LIN {X 0,Y 590.788,Z 779.363,A -85,B 0,C 180,E1 25957.461,E2 25957.461} C_VEL
LIN {X 0,Y 599.136,Z 539.916,A -85,B 0,C 180,E1 25954.035,E2 25954.035} C_VEL
LIN {X 0,Y 604.278,Z 401.411,A -85,B 0,C 180,E1 25952.028,E2 25952.028} C_VEL
LIN {X 0,Y 593.567,Z 385.03,A -85,B 0,C 180,E1 25950.244,E2 25950.244} C_VEL
LIN {X 0,Y 582.771,Z 369.958,A -85,B 0,C 180,E1 25948.293,E2 25948.293} C_VEL
LIN {X 0,Y 574.753,Z 359.34,A -85,B 0,C 180,E1 25946.725,E2 25946.725} C_VEL
LIN {X 0,Y 565.367,Z 346.989,A -85,B 0,C 180,E1 25944.67,E2 25944.67} C_VEL
LIN {X 0,Y 561.776,Z 340.566,A -85,B 0,C 180,E1 25943.052,E2 25943.052} C_VEL
LIN {X 0,Y 559.747,Z 336.589,A -85,B 0,C 180,E1 25942.032,E2 25942.032} C_VEL
LIN {X 0,Y 557.15,Z 331.806,A -85,B 0,C 180,E1 25940.705,E2 25940.705} C_VEL
LIN {X 0,Y 555.047,Z 327.971,A -85,B 0,C 180,E1 25939.577,E2 25939.577} C_VEL
LIN {X 0,Y 552.236,Z 323.289,A -85,B 0,C 180,E1 25938.036,E2 25938.036} C_VEL
LIN {X 0,Y 551.411,Z 321.689,A -85,B 0,C 180,E1 25937.519,E2 25937.519} C_VEL
LIN {X 0,Y 549.142,Z 318.092,A -85,B 0,C 180,E1 25936.176,E2 25936.176} C_VEL
LIN {X 0,Y 548.449,Z 316.544,A -85,B 0,C 180,E1 25935.654,E2 25935.654} C_VEL
LIN {X 0,Y 545.984,Z 313.041,A -85,B 0,C 180,E1 25934.097,E2 25934.097} C_VEL
LIN {X 0,Y 545.58,Z 311.452,A -85,B 0,C 180,E1 25933.459,E2 25933.459} C_VEL
LIN {X 0,Y 545.545,Z 311.25,A -85,B 0,C 180,E1 25930.241,E2 25930.241} C_VEL
LIN {X 0,Y 545.551,Z 311.212,A -85,B 0,C 180,E1 25926.842,E2 25926.842} C_VEL
LIN {X 0,Y 545.55,Z 311.247,A -85,B 0,C 180,E1 25923.362,E2 25923.362} C_VEL
LIN {X 0,Y 545.546,Z 311.235,A -85,B 0,C 180,E1 25920,E2 25920} C_VEL
LIN {X 0,Y 545.545,Z 311.216,A -85,B 0,C 180,E1 25916.743,E2 25916.743} C_VEL
LIN {X 0,Y 545.564,Z 311.275,A -85,B 0,C 180,E1 25913.264,E2 25913.264} C_VEL
LIN {X 0,Y 545.547,Z 311.219,A -85,B 0,C 180,E1 25909.799,E2 25909.799} C_VEL
LIN {X 0,Y 545.543,Z 311.229,A -85,B 0,C 180,E1 25906.54,E2 25906.54} C_VEL
LIN {X 0,Y 545.559,Z 311.26,A -85,B 0,C 180,E1 25903.167,E2 25903.167} C_VEL
LIN {X 0,Y 545.63,Z 311.708,A -85,B 0,C 180,E1 25901.945,E2 25901.945} C_VEL
LIN {X 0,Y 547.322,Z 315.338,A -85,B 0,C 180,E1 25900.58,E2 25900.58} C_VEL
LIN {X 0,Y 549.044,Z 317.373,A -85,B 0,C 180,E1 25899.645,E2 25899.645} C_VEL
LIN {X 0,Y 551.001,Z 321.182,A -85,B 0,C 180,E1 25898.384,E2 25898.384} C_VEL
LIN {X 0,Y 552.44,Z 323.078,A -85,B 0,C 180,E1 25897.661,E2 25897.661} C_VEL
LIN {X 0,Y 554.498,Z 326.812,A -85,B 0,C 180,E1 25896.515,E2 25896.515} C_VEL
LIN {X 0,Y 555.592,Z 328.37,A -85,B 0,C 180,E1 25896,E2 25896} C_VEL
LIN {X 0,Y 557.889,Z 332.375,A -85,B 0,C 180,E1 25894.864,E2 25894.864} C_VEL
LIN {X 0,Y 561.672,Z 339.042,A -85,B 0,C 180,E1 25893.107,E2 25893.107} C_VEL
LIN {X 0,Y 564.696,Z 344.498,A -85,B 0,C 180,E1 25891.786,E2 25891.786} C_VEL
LIN {X 0,Y 567.543,Z 349.518,A -85,B 0,C 180,E1 25890.674,E2 25890.674} C_VEL
LIN {X 0,Y 578.522,Z 363.571,A -85,B 0,C 180,E1 25888.391,E2 25888.391} C_VEL
LIN {X 0,Y 590.148,Z 379.589,A -85,B 0,C 180,E1 25886.239,E2 25886.239} C_VEL
LIN {X 0,Y 600.117,Z 394.544,A -85,B 0,C 180,E1 25884.532,E2 25884.532} C_VEL
LIN {X 0,Y 607.718,Z 406.774,A -85,B 0,C 180,E1 25883.311,E2 25883.311} C_VEL
LIN {X 0,Y 600.499,Z 616.97,A -85,B 0,C 180,E1 25880.226,E2 25880.226} C_VEL
LIN {X 0,Y 594.04,Z 824.716,A -85,B 0,C 180,E1 25877.25,E2 25877.25} C_VEL
LIN {X 0,Y 592.323,Z 852.282,A -85,B 0,C 180,E1 25876.741,E2 25876.741} C_VEL
LIN {X 0,Y 590.04,Z 878.41,A -85,B 0,C 180,E1 25876.074,E2 25876.074} C_VEL
LIN {X 0,Y 587.877,Z 899.594,A -85,B 0,C 180,E1 25875.411,E2 25875.411} C_VEL
LIN {X 0,Y 585.51,Z 920.264,A -85,B 0,C 180,E1 25874.645,E2 25874.645} C_VEL
LIN {X 0,Y 582.87,Z 941.326,A -85,B 0,C 180,E1 25873.734,E2 25873.734} C_VEL
LIN {X 0,Y 579.321,Z 967.03,A -85,B 0,C 180,E1 25872.441,E2 25872.441} C_VEL
LIN {X 0,Y 575.836,Z 989.761,A -85,B 0,C 180,E1 25871.096,E2 25871.096} C_VEL
LIN {X 0,Y 572.812,Z 1008.617,A -85,B 0,C 180,E1 25869.837,E2 25869.837} C_VEL
LIN {X 0,Y 569.828,Z 1026.571,A -85,B 0,C 180,E1 25868.5,E2 25868.5} C_VEL
LIN {X 0,Y 566.727,Z 1044.849,A -85,B 0,C 180,E1 25866.986,E2 25866.986} C_VEL
LIN {X 0,Y 564.355,Z 1058.093,A -85,B 0,C 180,E1 25865.761,E2 25865.761} C_VEL
LIN {X 0,Y 561.301,Z 1074.316,A -85,B 0,C 180,E1 25864.071,E2 25864.071} C_VEL
LIN {X 0,Y 557.893,Z 1092.847,A -85,B 0,C 180,E1 25861.918,E2 25861.918} C_VEL
LIN {X 0,Y 554.675,Z 1110.292,A -85,B 0,C 180,E1 25859.598,E2 25859.598} C_VEL
LIN {X 0,Y 552.277,Z 1124.437,A -85,B 0,C 180,E1 25857.483,E2 25857.483} C_VEL
LIN {X 0,Y 550.164,Z 1137.628,A -85,B 0,C 180,E1 25855.283,E2 25855.283} C_VEL
LIN {X 0,Y 548.084,Z 1152.164,A -85,B 0,C 180,E1 25852.526,E2 25852.526} C_VEL
LIN {X 0,Y 546.633,Z 1163.604,A -85,B 0,C 180,E1 25850.002,E2 25850.002} C_VEL
LIN {X 0,Y 545.65,Z 1172.702,A -85,B 0,C 180,E1 25847.709,E2 25847.709} C_VEL
LIN {X 0,Y 544.935,Z 1180.92,A -85,B 0,C 180,E1 25845.32,E2 25845.32} C_VEL
LIN {X 0,Y 544.377,Z 1189.025,A -85,B 0,C 180,E1 25842.517,E2 25842.517} C_VEL
LIN {X 0,Y 544.091,Z 1195.291,A -85,B 0,C 180,E1 25839.734,E2 25839.734} C_VEL
LIN {X 0,Y 543.978,Z 1199.369,A -85,B 0,C 180,E1 25837.392,E2 25837.392} C_VEL
LIN {X 0,Y 543.924,Z 1202.439,A -85,B 0,C 180,E1 25834.956,E2 25834.956} C_VEL
LIN {X 0,Y 543.91,Z 1204.495,A -85,B 0,C 180,E1 25832.212,E2 25832.212} C_VEL
LIN {X 0,Y 543.894,Z 1204.894,A -85,B 0,C 180,E1 25829.473,E2 25829.473} C_VEL
LIN {X 0,Y 543.915,Z 1204.043,A -85,B 0,C 180,E1 25827.05,E2 25827.05} C_VEL
LIN {X 0,Y 543.93,Z 1202.097,A -85,B 0,C 180,E1 25824.727,E2 25824.727} C_VEL
LIN {X 0,Y 543.984,Z 1198.889,A -85,B 0,C 180,E1 25822.289,E2 25822.289} C_VEL
LIN {X 0,Y 544.153,Z 1193.819,A -85,B 0,C 180,E1 25819.519,E2 25819.519} C_VEL
LIN {X 0,Y 544.513,Z 1186.94,A -85,B 0,C 180,E1 25816.717,E2 25816.717} C_VEL
LIN {X 0,Y 545.002,Z 1179.859,A -85,B 0,C 180,E1 25814.355,E2 25814.355} C_VEL
LIN {X 0,Y 545.737,Z 1171.893,A -85,B 0,C 180,E1 25812.074,E2 25812.074} C_VEL
LIN {X 0,Y 546.863,Z 1161.773,A -85,B 0,C 180,E1 25809.561,E2 25809.561} C_VEL
LIN {X 0,Y 548.605,Z 1148.289,A -85,B 0,C 180,E1 25806.703,E2 25806.703} C_VEL
LIN {X 0,Y 550.465,Z 1135.727,A -85,B 0,C 180,E1 25804.386,E2 25804.386} C_VEL
LIN {X 0,Y 552.556,Z 1122.677,A -85,B 0,C 180,E1 25802.238,E2 25802.238} C_VEL
LIN {X 0,Y 555.576,Z 1105.587,A -85,B 0,C 180,E1 25799.741,E2 25799.741} C_VEL
LIN {X 0,Y 558.686,Z 1088.219,A -85,B 0,C 180,E1 25797.527,E2 25797.527} C_VEL
LIN {X 0,Y 561.576,Z 1072.791,A -85,B 0,C 180,E1 25795.763,E2 25795.763} C_VEL
LIN {X 0,Y 564.688,Z 1056.271,A -85,B 0,C 180,E1 25794.058,E2 25794.058} C_VEL
LIN {X 0,Y 567.368,Z 1041.067,A -85,B 0,C 180,E1 25792.683,E2 25792.683} C_VEL
LIN {X 0,Y 571.091,Z 1019.418,A -85,B 0,C 180,E1 25790.929,E2 25790.929} C_VEL
LIN {X 0,Y 574.899,Z 996.123,A -85,B 0,C 180,E1 25789.293,E2 25789.293} C_VEL
LIN {X 0,Y 578.011,Z 976.204,A -85,B 0,C 180,E1 25788.061,E2 25788.061} C_VEL
LIN {X 0,Y 580.949,Z 956.254,A -85,B 0,C 180,E1 25786.968,E2 25786.968} C_VEL
LIN {X 0,Y 583.868,Z 935.058,A -85,B 0,C 180,E1 25785.952,E2 25785.952} C_VEL
LIN {X 0,Y 587.105,Z 909.113,A -85,B 0,C 180,E1 25784.89,E2 25784.89} C_VEL
LIN {X 0,Y 589.775,Z 883.656,A -85,B 0,C 180,E1 25784.048,E2 25784.048} C_VEL
LIN {X 0,Y 591.743,Z 862.08,A -85,B 0,C 180,E1 25783.464,E2 25783.464} C_VEL
LIN {X 0,Y 593.379,Z 840.414,A -85,B 0,C 180,E1 25782.996,E2 25782.996} C_VEL
LIN {X 0,Y 594.742,Z 814.677,A -85,B 0,C 180,E1 25782.568,E2 25782.568} C_VEL
LIN {X 0,Y 601.152,Z 593.035,A -85,B 0,C 180,E1 25779.439,E2 25779.439} C_VEL
LIN {X 0,Y 606.786,Z 406.521,A -85,B 0,C 180,E1 25776.755,E2 25776.755} C_VEL
LIN {X 0,Y 589.939,Z 382.189,A -85,B 0,C 180,E1 25774.39,E2 25774.39} C_VEL
LIN {X 0,Y 573.518,Z 359.446,A -85,B 0,C 180,E1 25771.888,E2 25771.888} C_VEL
LIN {X 0,Y 565.896,Z 348.958,A -85,B 0,C 180,E1 25770.589,E2 25770.589} C_VEL
LIN {X 0,Y 558.763,Z 335.53,A -85,B 0,C 180,E1 25768.192,E2 25768.192} C_VEL
LIN {X 0,Y 553.373,Z 325.76,A -85,B 0,C 180,E1 25766.276,E2 25766.276} C_VEL
LIN {X 0,Y 550.642,Z 320.898,A -85,B 0,C 180,E1 25765.26,E2 25765.26} C_VEL
LIN {X 0,Y 548.552,Z 317.065,A -85,B 0,C 180,E1 25764.442,E2 25764.442} C_VEL
LIN {X 0,Y 545.84,Z 312.595,A -85,B 0,C 180,E1 25763.405,E2 25763.405} C_VEL
LIN {X 0,Y 545.574,Z 311.357,A -85,B 0,C 180,E1 25763.074,E2 25763.074} C_VEL
LIN {X 0,Y 545.549,Z 311.245,A -85,B 0,C 180,E1 25759.709,E2 25759.709} C_VEL
LIN {X 0,Y 545.543,Z 311.204,A -85,B 0,C 180,E1 25756.395,E2 25756.395} C_VEL
LIN {X 0,Y 545.559,Z 311.271,A -85,B 0,C 180,E1 25753.028,E2 25753.028} C_VEL
LIN {X 0,Y 545.55,Z 311.196,A -85,B 0,C 180,E1 25749.592,E2 25749.592} C_VEL
LIN {X 0,Y 545.544,Z 311.275,A -85,B 0,C 180,E1 25746.208,E2 25746.208} C_VEL
LIN {X 0,Y 545.559,Z 311.277,A -85,B 0,C 180,E1 25742.77,E2 25742.77} C_VEL
LIN {X 0,Y 545.566,Z 311.272,A -85,B 0,C 180,E1 25739.37,E2 25739.37} C_VEL
LIN {X 0,Y 545.539,Z 311.278,A -85,B 0,C 180,E1 25736.006,E2 25736.006} C_VEL
LIN {X 0,Y 545.565,Z 311.267,A -85,B 0,C 180,E1 25732.629,E2 25732.629} C_VEL
LIN {X 0,Y 545.558,Z 311.268,A -85,B 0,C 180,E1 25729.216,E2 25729.216} C_VEL
LIN {X 0,Y 545.534,Z 311.267,A -85,B 0,C 180,E1 25725.825,E2 25725.825} C_VEL
LIN {X 0,Y 545.563,Z 311.258,A -85,B 0,C 180,E1 25722.508,E2 25722.508} C_VEL
LIN {X 0,Y 545.545,Z 311.261,A -85,B 0,C 180,E1 25719.172,E2 25719.172} C_VEL
LIN {X 0,Y 545.527,Z 311.212,A -85,B 0,C 180,E1 25715.759,E2 25715.759} C_VEL
LIN {X 0,Y 545.566,Z 311.254,A -85,B 0,C 180,E1 25712.374,E2 25712.374} C_VEL
LIN {X 0,Y 545.524,Z 311.209,A -85,B 0,C 180,E1 25709.067,E2 25709.067} C_VEL
LIN {X 0,Y 545.531,Z 311.278,A -85,B 0,C 180,E1 25705.565,E2 25705.565} C_VEL
LIN {X 0,Y 545.573,Z 311.483,A -85,B 0,C 180,E1 25702.673,E2 25702.673} C_VEL
LIN {X 0,Y 547.112,Z 315.058,A -85,B 0,C 180,E1 25701.85,E2 25701.85} C_VEL
LIN {X 0,Y 548.285,Z 316.8,A -85,B 0,C 180,E1 25701.413,E2 25701.413} C_VEL
LIN {X 0,Y 550.113,Z 320.411,A -85,B 0,C 180,E1 25700.628,E2 25700.628} C_VEL
LIN {X 0,Y 551.214,Z 322.439,A -85,B 0,C 180,E1 25700.183,E2 25700.183} C_VEL
LIN {X 0,Y 554.259,Z 328.328,A -85,B 0,C 180,E1 25698.954,E2 25698.954} C_VEL
LIN {X 0,Y 556.098,Z 331.679,A -85,B 0,C 180,E1 25698.259,E2 25698.259} C_VEL
LIN {X 0,Y 562.517,Z 344.33,A -85,B 0,C 180,E1 25695.83,E2 25695.83} C_VEL
LIN {X 0,Y 564.644,Z 348.18,A -85,B 0,C 180,E1 25695.187,E2 25695.187} C_VEL
LIN {X 0,Y 579.441,Z 368.707,A -85,B 0,C 180,E1 25692.811,E2 25692.811} C_VEL
LIN {X 0,Y 594.651,Z 390.663,A -85,B 0,C 180,E1 25690.574,E2 25690.574} C_VEL
LIN {X 0,Y 601.282,Z 400.794,A -85,B 0,C 180,E1 25689.652,E2 25689.652} C_VEL
LIN {X 0,Y 594.576,Z 614.61,A -85,B 0,C 180,E1 25686.64,E2 25686.64} C_VEL
LIN {X 0,Y 593.661,Z 622.309,A -85,B 0,C 180,E1 25686.601,E2 25686.601} C_VEL
LIN {X 0,Y 588.726,Z 642.915,A -85,B 0,C 180,E1 25686.752,E2 25686.752} C_VEL
LIN {X 0,Y 587.972,Z 649.525,A -85,B 0,C 180,E1 25686.715,E2 25686.715} C_VEL
LIN {X 0,Y 583.597,Z 784.855,A -85,B 0,C 180,E1 25684.797,E2 25684.797} C_VEL
LIN {X 0,Y 581.939,Z 811.482,A -85,B 0,C 180,E1 25684.279,E2 25684.279} C_VEL
LIN {X 0,Y 579.838,Z 835.361,A -85,B 0,C 180,E1 25683.639,E2 25683.639} C_VEL
LIN {X 0,Y 577.586,Z 856.724,A -85,B 0,C 180,E1 25682.927,E2 25682.927} C_VEL
LIN {X 0,Y 574.452,Z 882.144,A -85,B 0,C 180,E1 25681.887,E2 25681.887} C_VEL
LIN {X 0,Y 571.387,Z 903.281,A -85,B 0,C 180,E1 25680.845,E2 25680.845} C_VEL
LIN {X 0,Y 568.337,Z 922.57,A -85,B 0,C 180,E1 25679.743,E2 25679.743} C_VEL
LIN {X 0,Y 564.588,Z 944.778,A -85,B 0,C 180,E1 25678.277,E2 25678.277} C_VEL
LIN {X 0,Y 560.871,Z 964.796,A -85,B 0,C 180,E1 25676.727,E2 25676.727} C_VEL
LIN {X 0,Y 557.656,Z 981.532,A -85,B 0,C 180,E1 25675.26,E2 25675.26} C_VEL
LIN {X 0,Y 553.995,Z 1000.37,A -85,B 0,C 180,E1 25673.394,E2 25673.394} C_VEL
LIN {X 0,Y 550.34,Z 1018.522,A -85,B 0,C 180,E1 25671.307,E2 25671.307} C_VEL
LIN {X 0,Y 547.515,Z 1033.091,A -85,B 0,C 180,E1 25669.412,E2 25669.412} C_VEL
LIN {X 0,Y 544.571,Z 1048.925,A -85,B 0,C 180,E1 25667.084,E2 25667.084} C_VEL
LIN {X 0,Y 542.122,Z 1062.63,A -85,B 0,C 180,E1 25664.745,E2 25664.745} C_VEL
LIN {X 0,Y 540.353,Z 1073.663,A -85,B 0,C 180,E1 25662.612,E2 25662.612} C_VEL
LIN {X 0,Y 538.583,Z 1086.085,A -85,B 0,C 180,E1 25659.834,E2 25659.834} C_VEL
LIN {X 0,Y 537.402,Z 1096.194,A -85,B 0,C 180,E1 25657.161,E2 25657.161} C_VEL
LIN {X 0,Y 536.685,Z 1105.073,A -85,B 0,C 180,E1 25654.488,E2 25654.488} C_VEL
LIN {X 0,Y 536.258,Z 1111.875,A -85,B 0,C 180,E1 25651.923,E2 25651.923} C_VEL
LIN {X 0,Y 536.038,Z 1116.676,A -85,B 0,C 180,E1 25649.679,E2 25649.679} C_VEL
LIN {X 0,Y 535.95,Z 1120.549,A -85,B 0,C 180,E1 25647.327,E2 25647.327} C_VEL
LIN {X 0,Y 535.903,Z 1123.56,A -85,B 0,C 180,E1 25644.54,E2 25644.54} C_VEL
LIN {X 0,Y 535.915,Z 1124.748,A -85,B 0,C 180,E1 25642.172,E2 25642.172} C_VEL
LIN {X 0,Y 535.897,Z 1124.806,A -85,B 0,C 180,E1 25640.008,E2 25640.008} C_VEL
LIN {X 0,Y 535.914,Z 1123.784,A -85,B 0,C 180,E1 25637.72,E2 25637.72} C_VEL
LIN {X 0,Y 535.927,Z 1121.277,A -85,B 0,C 180,E1 25635.08,E2 25635.08} C_VEL
LIN {X 0,Y 536.034,Z 1117.021,A -85,B 0,C 180,E1 25632.412,E2 25632.412} C_VEL
LIN {X 0,Y 536.241,Z 1112.285,A -85,B 0,C 180,E1 25630.163,E2 25630.163} C_VEL
LIN {X 0,Y 536.603,Z 1106.05,A -85,B 0,C 180,E1 25627.775,E2 25627.775} C_VEL
LIN {X 0,Y 537.359,Z 1096.738,A -85,B 0,C 180,E1 25624.898,E2 25624.898} C_VEL
LIN {X 0,Y 538.514,Z 1086.699,A -85,B 0,C 180,E1 25622.223,E2 25622.223} C_VEL
LIN {X 0,Y 540.316,Z 1074.141,A -85,B 0,C 180,E1 25619.375,E2 25619.375} C_VEL
LIN {X 0,Y 542.16,Z 1062.795,A -85,B 0,C 180,E1 25617.167,E2 25617.167} C_VEL
LIN {X 0,Y 544.698,Z 1048.834,A -85,B 0,C 180,E1 25614.774,E2 25614.774} C_VEL
LIN {X 0,Y 547.719,Z 1032.714,A -85,B 0,C 180,E1 25612.4,E2 25612.4} C_VEL
LIN {X 0,Y 550.595,Z 1018.237,A -85,B 0,C 180,E1 25610.517,E2 25610.517} C_VEL
LIN {X 0,Y 554.342,Z 999.904,A -85,B 0,C 180,E1 25608.413,E2 25608.413} C_VEL
LIN {X 0,Y 557.857,Z 982.219,A -85,B 0,C 180,E1 25606.65,E2 25606.65} C_VEL
LIN {X 0,Y 561.158,Z 965.503,A -85,B 0,C 180,E1 25605.168,E2 25605.168} C_VEL
LIN {X 0,Y 565.097,Z 945.093,A -85,B 0,C 180,E1 25603.568,E2 25603.568} C_VEL
LIN {X 0,Y 569.057,Z 922.587,A -85,B 0,C 180,E1 25602.068,E2 25602.068} C_VEL
LIN {X 0,Y 572.335,Z 902.847,A -85,B 0,C 180,E1 25600.93,E2 25600.93} C_VEL
LIN {X 0,Y 576.001,Z 878.581,A -85,B 0,C 180,E1 25599.737,E2 25599.737} C_VEL
LIN {X 0,Y 578.96,Z 855.49,A -85,B 0,C 180,E1 25598.807,E2 25598.807} C_VEL
LIN {X 0,Y 581.4,Z 833.425,A -85,B 0,C 180,E1 25598.073,E2 25598.073} C_VEL
LIN {X 0,Y 583.848,Z 805.824,A -85,B 0,C 180,E1 25597.362,E2 25597.362} C_VEL
LIN {X 0,Y 585.261,Z 783.212,A -85,B 0,C 180,E1 25596.937,E2 25596.937} C_VEL
LIN {X 0,Y 593.876,Z 548.322,A -85,B 0,C 180,E1 25593.549,E2 25593.549} C_VEL
LIN {X 0,Y 599.32,Z 405.367,A -85,B 0,C 180,E1 25591.452,E2 25591.452} C_VEL
LIN {X 0,Y 589.748,Z 390.74,A -85,B 0,C 180,E1 25589.815,E2 25589.815} C_VEL
LIN {X 0,Y 579.93,Z 376.804,A -85,B 0,C 180,E1 25587.996,E2 25587.996} C_VEL
LIN {X 0,Y 571.777,Z 365.901,A -85,B 0,C 180,E1 25586.371,E2 25586.371} C_VEL
LIN {X 0,Y 561.894,Z 353.19,A -85,B 0,C 180,E1 25584.216,E2 25584.216} C_VEL
LIN {X 0,Y 557.113,Z 347.152,A -85,B 0,C 180,E1 25583.033,E2 25583.033} C_VEL
LIN {X 0,Y 554.637,Z 342.483,A -85,B 0,C 180,E1 25581.8,E2 25581.8} C_VEL
LIN {X 0,Y 552.29,Z 338.046,A -85,B 0,C 180,E1 25580.562,E2 25580.562} C_VEL
LIN {X 0,Y 549.649,Z 333.261,A -85,B 0,C 180,E1 25579.114,E2 25579.114} C_VEL
LIN {X 0,Y 547.469,Z 329.509,A -85,B 0,C 180,E1 25577.869,E2 25577.869} C_VEL
LIN {X 0,Y 546.617,Z 327.981,A -85,B 0,C 180,E1 25577.348,E2 25577.348} C_VEL
LIN {X 0,Y 544.451,Z 324.327,A -85,B 0,C 180,E1 25575.991,E2 25575.991} C_VEL
LIN {X 0,Y 543.712,Z 322.903,A -85,B 0,C 180,E1 25575.465,E2 25575.465} C_VEL
LIN {X 0,Y 541.474,Z 319.601,A -85,B 0,C 180,E1 25573.999,E2 25573.999} C_VEL
LIN {X 0,Y 540.662,Z 317.663,A -85,B 0,C 180,E1 25573.257,E2 25573.257} C_VEL
LIN {X 0,Y 538.008,Z 313.901,A -85,B 0,C 180,E1 25571.253,E2 25571.253} C_VEL
LIN {X 0,Y 537.637,Z 312.424,A -85,B 0,C 180,E1 25570.501,E2 25570.501} C_VEL
LIN {X 0,Y 537.606,Z 312.2,A -85,B 0,C 180,E1 25567.158,E2 25567.158} C_VEL
LIN {X 0,Y 537.616,Z 312.248,A -85,B 0,C 180,E1 25563.732,E2 25563.732} C_VEL
LIN {X 0,Y 537.61,Z 312.215,A -85,B 0,C 180,E1 25560.213,E2 25560.213} C_VEL
LIN {X 0,Y 537.604,Z 312.206,A -85,B 0,C 180,E1 25556.908,E2 25556.908} C_VEL
LIN {X 0,Y 537.622,Z 312.262,A -85,B 0,C 180,E1 25553.486,E2 25553.486} C_VEL
LIN {X 0,Y 537.613,Z 312.201,A -85,B 0,C 180,E1 25550.04,E2 25550.04} C_VEL
LIN {X 0,Y 537.603,Z 312.219,A -85,B 0,C 180,E1 25546.666,E2 25546.666} C_VEL
LIN {X 0,Y 537.678,Z 312.682,A -85,B 0,C 180,E1 25544.861,E2 25544.861} C_VEL
LIN {X 0,Y 539.663,Z 316.679,A -85,B 0,C 180,E1 25542.978,E2 25542.978} C_VEL
LIN {X 0,Y 541.191,Z 318.389,A -85,B 0,C 180,E1 25542.028,E2 25542.028} C_VEL
LIN {X 0,Y 543.193,Z 322.266,A -85,B 0,C 180,E1 25540.538,E2 25540.538} C_VEL
LIN {X 0,Y 544.676,Z 324.196,A -85,B 0,C 180,E1 25539.699,E2 25539.699} C_VEL
LIN {X 0,Y 546.678,Z 327.904,A -85,B 0,C 180,E1 25538.43,E2 25538.43} C_VEL
LIN {X 0,Y 547.899,Z 329.537,A -85,B 0,C 180,E1 25537.805,E2 25537.805} C_VEL
LIN {X 0,Y 550.16,Z 333.541,A -85,B 0,C 180,E1 25536.545,E2 25536.545} C_VEL
LIN {X 0,Y 551.166,Z 335.27,A -85,B 0,C 180,E1 25536.023,E2 25536.023} C_VEL
LIN {X 0,Y 554.132,Z 340.375,A -85,B 0,C 180,E1 25534.567,E2 25534.567} C_VEL
LIN {X 0,Y 557.254,Z 346.035,A -85,B 0,C 180,E1 25533.094,E2 25533.094} C_VEL
LIN {X 0,Y 559.701,Z 349.915,A -85,B 0,C 180,E1 25532.155,E2 25532.155} C_VEL
LIN {X 0,Y 569.252,Z 362.11,A -85,B 0,C 180,E1 25530.018,E2 25530.018} C_VEL
LIN {X 0,Y 576.839,Z 372.123,A -85,B 0,C 180,E1 25528.463,E2 25528.463} C_VEL
LIN {X 0,Y 586.146,Z 384.955,A -85,B 0,C 180,E1 25526.708,E2 25526.708} C_VEL
LIN {X 0,Y 596.346,Z 400.335,A -85,B 0,C 180,E1 25524.922,E2 25524.922} C_VEL
LIN {X 0,Y 602.725,Z 411.033,A -85,B 0,C 180,E1 25523.856,E2 25523.856} C_VEL
LIN {X 0,Y 595.171,Z 619.586,A -85,B 0,C 180,E1 25520.771,E2 25520.771} C_VEL
LIN {X 0,Y 588.394,Z 823.949,A -85,B 0,C 180,E1 25517.812,E2 25517.812} C_VEL
LIN {X 0,Y 586.619,Z 851.271,A -85,B 0,C 180,E1 25517.306,E2 25517.306} C_VEL
LIN {X 0,Y 584.167,Z 877.942,A -85,B 0,C 180,E1 25516.622,E2 25516.622} C_VEL
LIN {X 0,Y 581.868,Z 899.303,A -85,B 0,C 180,E1 25515.948,E2 25515.948} C_VEL
LIN {X 0,Y 579.397,Z 919.967,A -85,B 0,C 180,E1 25515.175,E2 25515.175} C_VEL
LIN {X 0,Y 576.483,Z 942.167,A -85,B 0,C 180,E1 25514.205,E2 25514.205} C_VEL
LIN {X 0,Y 572.541,Z 969.084,A -85,B 0,C 180,E1 25512.82,E2 25512.82} C_VEL
LIN {X 0,Y 569.29,Z 989.489,A -85,B 0,C 180,E1 25511.597,E2 25511.597} C_VEL
LIN {X 0,Y 566.28,Z 1007.447,A -85,B 0,C 180,E1 25510.391,E2 25510.391} C_VEL
LIN {X 0,Y 563.043,Z 1026.1,A -85,B 0,C 180,E1 25508.992,E2 25508.992} C_VEL
LIN {X 0,Y 559.678,Z 1045.078,A -85,B 0,C 180,E1 25507.402,E2 25507.402} C_VEL
LIN {X 0,Y 555.65,Z 1067.446,A -85,B 0,C 180,E1 25505.283,E2 25505.283} C_VEL
LIN {X 0,Y 552.541,Z 1083.586,A -85,B 0,C 180,E1 25503.499,E2 25503.499} C_VEL
LIN {X 0,Y 549.554,Z 1098.822,A -85,B 0,C 180,E1 25501.6,E2 25501.6} C_VEL
LIN {X 0,Y 546.949,Z 1112.601,A -85,B 0,C 180,E1 25499.697,E2 25499.697} C_VEL
LIN {X 0,Y 544.608,Z 1125.771,A -85,B 0,C 180,E1 25497.677,E2 25497.677} C_VEL
LIN {X 0,Y 542.106,Z 1140.846,A -85,B 0,C 180,E1 25495.091,E2 25495.091} C_VEL
LIN {X 0,Y 540.078,Z 1154.228,A -85,B 0,C 180,E1 25492.419,E2 25492.419} C_VEL
LIN {X 0,Y 538.721,Z 1164.52,A -85,B 0,C 180,E1 25490.082,E2 25490.082} C_VEL
LIN {X 0,Y 537.701,Z 1173.511,A -85,B 0,C 180,E1 25487.756,E2 25487.756} C_VEL
LIN {X 0,Y 536.844,Z 1183.174,A -85,B 0,C 180,E1 25484.837,E2 25484.837} C_VEL
LIN {X 0,Y 536.324,Z 1190.568,A -85,B 0,C 180,E1 25482.052,E2 25482.052} C_VEL
LIN {X 0,Y 536.091,Z 1195.702,A -85,B 0,C 180,E1 25479.663,E2 25479.663} C_VEL
LIN {X 0,Y 535.978,Z 1199.686,A -85,B 0,C 180,E1 25477.288,E2 25477.288} C_VEL
LIN {X 0,Y 535.918,Z 1202.89,A -85,B 0,C 180,E1 25474.602,E2 25474.602} C_VEL
LIN {X 0,Y 535.908,Z 1204.645,A -85,B 0,C 180,E1 25471.711,E2 25471.711} C_VEL
LIN {X 0,Y 535.899,Z 1204.849,A -85,B 0,C 180,E1 25469.252,E2 25469.252} C_VEL
LIN {X 0,Y 535.916,Z 1203.972,A -85,B 0,C 180,E1 25466.899,E2 25466.899} C_VEL
LIN {X 0,Y 535.932,Z 1201.98,A -85,B 0,C 180,E1 25464.54,E2 25464.54} C_VEL
LIN {X 0,Y 536,Z 1198.727,A -85,B 0,C 180,E1 25462.066,E2 25462.066} C_VEL
LIN {X 0,Y 536.184,Z 1193.351,A -85,B 0,C 180,E1 25459.144,E2 25459.144} C_VEL
LIN {X 0,Y 536.58,Z 1186.673,A -85,B 0,C 180,E1 25456.421,E2 25456.421} C_VEL
LIN {X 0,Y 537.084,Z 1179.858,A -85,B 0,C 180,E1 25454.118,E2 25454.118} C_VEL
LIN {X 0,Y 537.886,Z 1171.844,A -85,B 0,C 180,E1 25451.79,E2 25451.79} C_VEL
LIN {X 0,Y 539.073,Z 1161.773,A -85,B 0,C 180,E1 25449.252,E2 25449.252} C_VEL
LIN {X 0,Y 540.935,Z 1148.287,A -85,B 0,C 180,E1 25446.353,E2 25446.353} C_VEL
LIN {X 0,Y 542.817,Z 1136.36,A -85,B 0,C 180,E1 25444.116,E2 25444.116} C_VEL
LIN {X 0,Y 545.002,Z 1123.401,A -85,B 0,C 180,E1 25441.942,E2 25441.942} C_VEL
LIN {X 0,Y 548.028,Z 1107.206,A -85,B 0,C 180,E1 25439.523,E2 25439.523} C_VEL
LIN {X 0,Y 551.436,Z 1089.143,A -85,B 0,C 180,E1 25437.17,E2 25437.17} C_VEL
LIN {X 0,Y 554.455,Z 1073.791,A -85,B 0,C 180,E1 25435.386,E2 25435.386} C_VEL
LIN {X 0,Y 557.399,Z 1057.659,A -85,B 0,C 180,E1 25433.753,E2 25433.753} C_VEL
LIN {X 0,Y 560.701,Z 1039.495,A -85,B 0,C 180,E1 25432.097,E2 25432.097} C_VEL
LIN {X 0,Y 564.767,Z 1016.991,A -85,B 0,C 180,E1 25430.275,E2 25430.275} C_VEL
LIN {X 0,Y 568.503,Z 995.044,A -85,B 0,C 180,E1 25428.736,E2 25428.736} C_VEL
LIN {X 0,Y 571.646,Z 975.751,A -85,B 0,C 180,E1 25427.535,E2 25427.535} C_VEL
LIN {X 0,Y 574.662,Z 956.079,A -85,B 0,C 180,E1 25426.449,E2 25426.449} C_VEL
LIN {X 0,Y 577.695,Z 934.913,A -85,B 0,C 180,E1 25425.426,E2 25425.426} C_VEL
LIN {X 0,Y 581.073,Z 909.085,A -85,B 0,C 180,E1 25424.361,E2 25424.361} C_VEL
LIN {X 0,Y 583.89,Z 883.362,A -85,B 0,C 180,E1 25423.505,E2 25423.505} C_VEL
LIN {X 0,Y 585.934,Z 861.677,A -85,B 0,C 180,E1 25422.916,E2 25422.916} C_VEL
LIN {X 0,Y 587.637,Z 839.987,A -85,B 0,C 180,E1 25422.446,E2 25422.446} C_VEL
LIN {X 0,Y 589.051,Z 813.903,A -85,B 0,C 180,E1 25422.012,E2 25422.012} C_VEL
LIN {X 0,Y 595.73,Z 591.408,A -85,B 0,C 180,E1 25418.853,E2 25418.853} C_VEL
LIN {X 0,Y 601.394,Z 410.5,A -85,B 0,C 180,E1 25416.233,E2 25416.233} C_VEL
LIN {X 0,Y 585.583,Z 387.534,A -85,B 0,C 180,E1 25413.972,E2 25413.972} C_VEL
LIN {X 0,Y 569.733,Z 365.449,A -85,B 0,C 180,E1 25411.504,E2 25411.504} C_VEL
LIN {X 0,Y 558.536,Z 350.402,A -85,B 0,C 180,E1 25409.61,E2 25409.61} C_VEL
LIN {X 0,Y 556.75,Z 347.357,A -85,B 0,C 180,E1 25409.124,E2 25409.124} C_VEL
LIN {X 0,Y 550.385,Z 335.715,A -85,B 0,C 180,E1 25406.895,E2 25406.895} C_VEL
LIN {X 0,Y 547.905,Z 331.185,A -85,B 0,C 180,E1 25405.976,E2 25405.976} C_VEL
LIN {X 0,Y 545.49,Z 326.8,A -85,B 0,C 180,E1 25405.051,E2 25405.051} C_VEL
LIN {X 0,Y 542.659,Z 321.839,A -85,B 0,C 180,E1 25403.952,E2 25403.952} C_VEL
LIN {X 0,Y 540.613,Z 317.903,A -85,B 0,C 180,E1 25403.086,E2 25403.086} C_VEL
LIN {X 0,Y 537.991,Z 313.794,A -85,B 0,C 180,E1 25402.051,E2 25402.051} C_VEL
LIN {X 0,Y 537.636,Z 312.416,A -85,B 0,C 180,E1 25401.722,E2 25401.722} C_VEL
LIN {X 0,Y 537.613,Z 312.253,A -85,B 0,C 180,E1 25398.432,E2 25398.432} C_VEL
LIN {X 0,Y 537.619,Z 312.194,A -85,B 0,C 180,E1 25394.982,E2 25394.982} C_VEL
LIN {X 0,Y 537.614,Z 312.222,A -85,B 0,C 180,E1 25391.588,E2 25391.588} C_VEL
LIN {X 0,Y 537.6,Z 312.202,A -85,B 0,C 180,E1 25388.234,E2 25388.234} C_VEL
LIN {X 0,Y 537.618,Z 312.245,A -85,B 0,C 180,E1 25384.908,E2 25384.908} C_VEL
LIN {X 0,Y 537.621,Z 312.246,A -85,B 0,C 180,E1 25381.492,E2 25381.492} C_VEL
LIN {X 0,Y 537.6,Z 312.248,A -85,B 0,C 180,E1 25378.081,E2 25378.081} C_VEL
LIN {X 0,Y 537.621,Z 312.249,A -85,B 0,C 180,E1 25374.664,E2 25374.664} C_VEL
LIN {X 0,Y 537.623,Z 312.253,A -85,B 0,C 180,E1 25371.228,E2 25371.228} C_VEL
LIN {X 0,Y 537.598,Z 312.259,A -85,B 0,C 180,E1 25367.868,E2 25367.868} C_VEL
LIN {X 0,Y 537.625,Z 312.256,A -85,B 0,C 180,E1 25364.441,E2 25364.441} C_VEL
LIN {X 0,Y 537.621,Z 312.261,A -85,B 0,C 180,E1 25361.006,E2 25361.006} C_VEL
LIN {X 0,Y 537.591,Z 312.263,A -85,B 0,C 180,E1 25357.586,E2 25357.586} C_VEL
LIN {X 0,Y 537.614,Z 312.187,A -85,B 0,C 180,E1 25354.177,E2 25354.177} C_VEL
LIN {X 0,Y 537.611,Z 312.242,A -85,B 0,C 180,E1 25350.837,E2 25350.837} C_VEL
LIN {X 0,Y 537.58,Z 312.206,A -85,B 0,C 180,E1 25347.41,E2 25347.41} C_VEL
LIN {X 0,Y 537.656,Z 312.464,A -85,B 0,C 180,E1 25344.072,E2 25344.072} C_VEL
LIN {X 0,Y 539.172,Z 316.09,A -85,B 0,C 180,E1 25343.201,E2 25343.201} C_VEL
LIN {X 0,Y 540.569,Z 318.17,A -85,B 0,C 180,E1 25342.648,E2 25342.648} C_VEL
LIN {X 0,Y 543.392,Z 323.586,A -85,B 0,C 180,E1 25341.406,E2 25341.406} C_VEL
LIN {X 0,Y 545.853,Z 328.013,A -85,B 0,C 180,E1 25340.397,E2 25340.397} C_VEL
LIN {X 0,Y 550.857,Z 337.713,A -85,B 0,C 180,E1 25338.368,E2 25338.368} C_VEL
LIN {X 0,Y 555.702,Z 347.351,A -85,B 0,C 180,E1 25336.509,E2 25336.509} C_VEL
LIN {X 0,Y 565.639,Z 360.717,A -85,B 0,C 180,E1 25334.786,E2 25334.786} C_VEL
LIN {X 0,Y 579.893,Z 380.779,A -85,B 0,C 180,E1 25332.52,E2 25332.52} C_VEL
LIN {X 0,Y 595.516,Z 403.747,A -85,B 0,C 180,E1 25330.241,E2 25330.241} C_VEL
LIN {X 0,Y 595.906,Z 404.854,A -85,B 0,C 180,E1 25330.177,E2 25330.177} C_VEL
LIN {X 0,Y 588.422,Z 635.331,A -85,B 0,C 180,E1 25326.914,E2 25326.914} C_VEL
LIN {X 0,Y 587.972,Z 649.525,A -85,B 0,C 180,E1 25326.715,E2 25326.715} C_VEL
LIN {X 0,Y 587.005,Z 657.229,A -85,B 0,C 180,E1 25326.681,E2 25326.681} C_VEL
LIN {X 0,Y 582.036,Z 677.827,A -85,B 0,C 180,E1 25326.834,E2 25326.834} C_VEL
LIN {X 0,Y 581.324,Z 684.43,A -85,B 0,C 180,E1 25326.792,E2 25326.792} C_VEL
LIN {X 0,Y 577.899,Z 785.614,A -85,B 0,C 180,E1 25325.347,E2 25325.347} C_VEL
LIN {X 0,Y 576.126,Z 812.71,A -85,B 0,C 180,E1 25324.81,E2 25324.81} C_VEL
LIN {X 0,Y 573.986,Z 836.194,A -85,B 0,C 180,E1 25324.175,E2 25324.175} C_VEL
LIN {X 0,Y 571.594,Z 858.136,A -85,B 0,C 180,E1 25323.436,E2 25323.436} C_VEL
LIN {X 0,Y 568.19,Z 884.448,A -85,B 0,C 180,E1 25322.341,E2 25322.341} C_VEL
LIN {X 0,Y 565.176,Z 904.485,A -85,B 0,C 180,E1 25321.34,E2 25321.34} C_VEL
LIN {X 0,Y 561.884,Z 924.579,A -85,B 0,C 180,E1 25320.179,E2 25320.179} C_VEL
LIN {X 0,Y 557.724,Z 947.925,A -85,B 0,C 180,E1 25318.598,E2 25318.598} C_VEL
LIN {X 0,Y 554.198,Z 966.252,A -85,B 0,C 180,E1 25317.158,E2 25317.158} C_VEL
LIN {X 0,Y 550.815,Z 983.204,A -85,B 0,C 180,E1 25315.654,E2 25315.654} C_VEL
LIN {X 0,Y 546.898,Z 1002.396,A -85,B 0,C 180,E1 25313.716,E2 25313.716} C_VEL
LIN {X 0,Y 543.279,Z 1019.553,A -85,B 0,C 180,E1 25311.711,E2 25311.711} C_VEL
LIN {X 0,Y 540.307,Z 1034.087,A -85,B 0,C 180,E1 25309.794,E2 25309.794} C_VEL
LIN {X 0,Y 537.072,Z 1050.489,A -85,B 0,C 180,E1 25307.33,E2 25307.33} C_VEL
LIN {X 0,Y 534.612,Z 1063.522,A -85,B 0,C 180,E1 25305.068,E2 25305.068} C_VEL
LIN {X 0,Y 532.66,Z 1075.054,A -85,B 0,C 180,E1 25302.797,E2 25302.797} C_VEL
LIN {X 0,Y 530.79,Z 1087.321,A -85,B 0,C 180,E1 25299.98,E2 25299.98} C_VEL
LIN {X 0,Y 529.7,Z 1095.828,A -85,B 0,C 180,E1 25297.683,E2 25297.683} C_VEL
LIN {X 0,Y 528.906,Z 1103.363,A -85,B 0,C 180,E1 25295.315,E2 25295.315} C_VEL
LIN {X 0,Y 528.308,Z 1111.443,A -85,B 0,C 180,E1 25292.278,E2 25292.278} C_VEL
LIN {X 0,Y 528.058,Z 1116.527,A -85,B 0,C 180,E1 25289.891,E2 25289.891} C_VEL
LIN {X 0,Y 527.961,Z 1120.273,A -85,B 0,C 180,E1 25287.612,E2 25287.612} C_VEL
LIN {X 0,Y 527.91,Z 1123.44,A -85,B 0,C 180,E1 25284.784,E2 25284.784} C_VEL
LIN {X 0,Y 527.915,Z 1124.754,A -85,B 0,C 180,E1 25282.162,E2 25282.162} C_VEL
LIN {X 0,Y 527.897,Z 1124.8,A -85,B 0,C 180,E1 25279.965,E2 25279.965} C_VEL
LIN {X 0,Y 527.913,Z 1123.835,A -85,B 0,C 180,E1 25277.753,E2 25277.753} C_VEL
LIN {X 0,Y 527.929,Z 1121.485,A -85,B 0,C 180,E1 25275.186,E2 25275.186} C_VEL
LIN {X 0,Y 528.032,Z 1117.391,A -85,B 0,C 180,E1 25272.478,E2 25272.478} C_VEL
LIN {X 0,Y 528.257,Z 1112.477,A -85,B 0,C 180,E1 25270.081,E2 25270.081} C_VEL
LIN {X 0,Y 528.735,Z 1105.432,A -85,B 0,C 180,E1 25267.308,E2 25267.308} C_VEL
LIN {X 0,Y 529.607,Z 1096.761,A -85,B 0,C 180,E1 25264.483,E2 25264.483} C_VEL
LIN {X 0,Y 530.692,Z 1088.239,A -85,B 0,C 180,E1 25262.144,E2 25262.144} C_VEL
LIN {X 0,Y 532.387,Z 1077.221,A -85,B 0,C 180,E1 25259.531,E2 25259.531} C_VEL
LIN {X 0,Y 534.502,Z 1064.686,A -85,B 0,C 180,E1 25257.019,E2 25257.019} C_VEL
LIN {X 0,Y 536.803,Z 1052.434,A -85,B 0,C 180,E1 25254.857,E2 25254.857} C_VEL
LIN {X 0,Y 540.088,Z 1036.135,A -85,B 0,C 180,E1 25252.344,E2 25252.344} C_VEL
LIN {X 0,Y 543.252,Z 1020.829,A -85,B 0,C 180,E1 25250.296,E2 25250.296} C_VEL
LIN {X 0,Y 546.786,Z 1004.342,A -85,B 0,C 180,E1 25248.341,E2 25248.341} C_VEL
LIN {X 0,Y 551.054,Z 984.217,A -85,B 0,C 180,E1 25246.267,E2 25246.267} C_VEL
LIN {X 0,Y 554.573,Z 967.254,A -85,B 0,C 180,E1 25244.736,E2 25244.736} C_VEL
LIN {X 0,Y 558.126,Z 949.644,A -85,B 0,C 180,E1 25243.326,E2 25243.326} C_VEL
LIN {X 0,Y 562.538,Z 926.371,A -85,B 0,C 180,E1 25241.711,E2 25241.711} C_VEL
LIN {X 0,Y 566.095,Z 905.927,A -85,B 0,C 180,E1 25240.504,E2 25240.504} C_VEL
LIN {X 0,Y 569.307,Z 885.847,A -85,B 0,C 180,E1 25239.479,E2 25239.479} C_VEL
LIN {X 0,Y 572.859,Z 860.69,A -85,B 0,C 180,E1 25238.402,E2 25238.402} C_VEL
LIN {X 0,Y 575.53,Z 837.91,A -85,B 0,C 180,E1 25237.613,E2 25237.613} C_VEL
LIN {X 0,Y 577.697,Z 815.914,A -85,B 0,C 180,E1 25236.999,E2 25236.999} C_VEL
LIN {X 0,Y 579.713,Z 788.632,A -85,B 0,C 180,E1 25236.429,E2 25236.429} C_VEL
LIN {X 0,Y 582.045,Z 730.67,A -85,B 0,C 180,E1 25235.571,E2 25235.571} C_VEL
LIN {X 0,Y 591.399,Z 488.055,A -85,B 0,C 180,E1 25232.051,E2 25232.051} C_VEL
LIN {X 0,Y 594.511,Z 409.438,A -85,B 0,C 180,E1 25230.881,E2 25230.881} C_VEL
LIN {X 0,Y 583.649,Z 392.867,A -85,B 0,C 180,E1 25228.945,E2 25228.945} C_VEL
LIN {X 0,Y 573.525,Z 378.756,A -85,B 0,C 180,E1 25226.983,E2 25226.983} C_VEL
LIN {X 0,Y 565.11,Z 367.508,A -85,B 0,C 180,E1 25225.213,E2 25225.213} C_VEL
LIN {X 0,Y 558.886,Z 359.665,A -85,B 0,C 180,E1 25223.793,E2 25223.793} C_VEL
LIN {X 0,Y 554.297,Z 353.953,A -85,B 0,C 180,E1 25222.68,E2 25222.68} C_VEL
LIN {X 0,Y 548.97,Z 347.3,A -85,B 0,C 180,E1 25221.251,E2 25221.251} C_VEL
LIN {X 0,Y 547.436,Z 344.284,A -85,B 0,C 180,E1 25220.418,E2 25220.418} C_VEL
LIN {X 0,Y 544.834,Z 339.532,A -85,B 0,C 180,E1 25218.956,E2 25218.956} C_VEL
LIN {X 0,Y 542.612,Z 335.362,A -85,B 0,C 180,E1 25217.59,E2 25217.59} C_VEL
LIN {X 0,Y 539.781,Z 330.572,A -85,B 0,C 180,E1 25215.801,E2 25215.801} C_VEL
LIN {X 0,Y 538.622,Z 328.846,A -85,B 0,C 180,E1 25215.064,E2 25215.064} C_VEL
LIN {X 0,Y 536.665,Z 325.242,A -85,B 0,C 180,E1 25213.577,E2 25213.577} C_VEL
LIN {X 0,Y 535.333,Z 323.37,A -85,B 0,C 180,E1 25212.623,E2 25212.623} C_VEL
LIN {X 0,Y 533.239,Z 319.434,A -85,B 0,C 180,E1 25210.698,E2 25210.698} C_VEL
LIN {X 0,Y 529.821,Z 314.038,A -85,B 0,C 180,E1 25207.046,E2 25207.046} C_VEL
LIN {X 0,Y 529.678,Z 313.298,A -85,B 0,C 180,E1 25206.068,E2 25206.068} C_VEL
LIN {X 0,Y 529.677,Z 313.196,A -85,B 0,C 180,E1 25202.597,E2 25202.597} C_VEL
LIN {X 0,Y 529.67,Z 313.241,A -85,B 0,C 180,E1 25199.135,E2 25199.135} C_VEL
LIN {X 0,Y 529.669,Z 313.186,A -85,B 0,C 180,E1 25195.669,E2 25195.669} C_VEL
LIN {X 0,Y 529.682,Z 313.208,A -85,B 0,C 180,E1 25192.188,E2 25192.188} C_VEL
LIN {X 0,Y 529.704,Z 313.444,A -85,B 0,C 180,E1 25189.009,E2 25189.009} C_VEL
LIN {X 0,Y 531.887,Z 317.785,A -85,B 0,C 180,E1 25186.076,E2 25186.076} C_VEL
LIN {X 0,Y 533.339,Z 319.501,A -85,B 0,C 180,E1 25184.895,E2 25184.895} C_VEL
LIN {X 0,Y 535.536,Z 323.573,A -85,B 0,C 180,E1 25182.954,E2 25182.954} C_VEL
LIN {X 0,Y 536.855,Z 325.158,A -85,B 0,C 180,E1 25182.103,E2 25182.103} C_VEL
LIN {X 0,Y 538.893,Z 328.985,A -85,B 0,C 180,E1 25180.602,E2 25180.602} C_VEL
LIN {X 0,Y 540.193,Z 330.642,A -85,B 0,C 180,E1 25179.862,E2 25179.862} C_VEL
LIN {X 0,Y 542.357,Z 334.626,A -85,B 0,C 180,E1 25178.477,E2 25178.477} C_VEL
LIN {X 0,Y 543.362,Z 335.993,A -85,B 0,C 180,E1 25177.951,E2 25177.951} C_VEL
LIN {X 0,Y 545.704,Z 340.137,A -85,B 0,C 180,E1 25176.628,E2 25176.628} C_VEL
LIN {X 0,Y 549.517,Z 346.854,A -85,B 0,C 180,E1 25174.684,E2 25174.684} C_VEL
LIN {X 0,Y 551.561,Z 350.135,A -85,B 0,C 180,E1 25173.863,E2 25173.863} C_VEL
LIN {X 0,Y 557.783,Z 357.823,A -85,B 0,C 180,E1 25172.307,E2 25172.307} C_VEL
LIN {X 0,Y 565.709,Z 367.847,A -85,B 0,C 180,E1 25170.511,E2 25170.511} C_VEL
LIN {X 0,Y 574.167,Z 379.168,A -85,B 0,C 180,E1 25168.738,E2 25168.738} C_VEL
LIN {X 0,Y 583.219,Z 391.854,A -85,B 0,C 180,E1 25166.991,E2 25166.991} C_VEL
LIN {X 0,Y 593.027,Z 406.837,A -85,B 0,C 180,E1 25165.242,E2 25165.242} C_VEL
LIN {X 0,Y 597.824,Z 415.116,A -85,B 0,C 180,E1 25164.415,E2 25164.415} C_VEL
LIN {X 0,Y 589.845,Z 624.272,A -85,B 0,C 180,E1 25161.298,E2 25161.298} C_VEL
LIN {X 0,Y 582.839,Z 823.699,A -85,B 0,C 180,E1 25158.381,E2 25158.381} C_VEL
LIN {X 0,Y 580.951,Z 851.157,A -85,B 0,C 180,E1 25157.867,E2 25157.867} C_VEL
LIN {X 0,Y 578.419,Z 877.365,A -85,B 0,C 180,E1 25157.191,E2 25157.191} C_VEL
LIN {X 0,Y 576.023,Z 898.61,A -85,B 0,C 180,E1 25156.516,E2 25156.516} C_VEL
LIN {X 0,Y 573.349,Z 919.814,A -85,B 0,C 180,E1 25155.714,E2 25155.714} C_VEL
LIN {X 0,Y 570.25,Z 942.2,A -85,B 0,C 180,E1 25154.726,E2 25154.726} C_VEL
LIN {X 0,Y 566.15,Z 968.929,A -85,B 0,C 180,E1 25153.335,E2 25153.335} C_VEL
LIN {X 0,Y 562.8,Z 989.081,A -85,B 0,C 180,E1 25152.118,E2 25152.118} C_VEL
LIN {X 0,Y 559.526,Z 1007.811,A -85,B 0,C 180,E1 25150.846,E2 25150.846} C_VEL
LIN {X 0,Y 556.203,Z 1026.137,A -85,B 0,C 180,E1 25149.455,E2 25149.455} C_VEL
LIN {X 0,Y 552.456,Z 1046.449,A -85,B 0,C 180,E1 25147.727,E2 25147.727} C_VEL
LIN {X 0,Y 548.232,Z 1068.682,A -85,B 0,C 180,E1 25145.567,E2 25145.567} C_VEL
LIN {X 0,Y 544.974,Z 1085.823,A -85,B 0,C 180,E1 25143.683,E2 25143.683} C_VEL
LIN {X 0,Y 542.745,Z 1097.336,A -85,B 0,C 180,E1 25142.262,E2 25142.262} C_VEL
LIN {X 0,Y 539.819,Z 1111.828,A -85,B 0,C 180,E1 25140.252,E2 25140.252} C_VEL
LIN {X 0,Y 537.291,Z 1125.068,A -85,B 0,C 180,E1 25138.208,E2 25138.208} C_VEL
LIN {X 0,Y 534.856,Z 1138.893,A -85,B 0,C 180,E1 25135.822,E2 25135.822} C_VEL
LIN {X 0,Y 532.454,Z 1153.711,A -85,B 0,C 180,E1 25132.874,E2 25132.874} C_VEL
LIN {X 0,Y 530.995,Z 1164.06,A -85,B 0,C 180,E1 25130.502,E2 25130.502} C_VEL
LIN {X 0,Y 529.89,Z 1173.105,A -85,B 0,C 180,E1 25128.14,E2 25128.14} C_VEL
LIN {X 0,Y 529.005,Z 1182.071,A -85,B 0,C 180,E1 25125.426,E2 25125.426} C_VEL
LIN {X 0,Y 528.384,Z 1190.059,A -85,B 0,C 180,E1 25122.456,E2 25122.456} C_VEL
LIN {X 0,Y 528.113,Z 1195.492,A -85,B 0,C 180,E1 25119.921,E2 25119.921} C_VEL
LIN {X 0,Y 527.983,Z 1199.523,A -85,B 0,C 180,E1 25117.508,E2 25117.508} C_VEL
LIN {X 0,Y 527.926,Z 1202.581,A -85,B 0,C 180,E1 25114.965,E2 25114.965} C_VEL
LIN {X 0,Y 527.911,Z 1204.577,A -85,B 0,C 180,E1 25112.062,E2 25112.062} C_VEL
LIN {X 0,Y 527.896,Z 1204.871,A -85,B 0,C 180,E1 25109.349,E2 25109.349} C_VEL
LIN {X 0,Y 527.916,Z 1204.037,A -85,B 0,C 180,E1 25106.96,E2 25106.96} C_VEL
LIN {X 0,Y 527.932,Z 1202.091,A -85,B 0,C 180,E1 25104.566,E2 25104.566} C_VEL
LIN {X 0,Y 527.994,Z 1199.043,A -85,B 0,C 180,E1 25102.164,E2 25102.164} C_VEL
LIN {X 0,Y 528.171,Z 1194.253,A -85,B 0,C 180,E1 25099.419,E2 25099.419} C_VEL
LIN {X 0,Y 528.591,Z 1187.276,A -85,B 0,C 180,E1 25096.435,E2 25096.435} C_VEL
LIN {X 0,Y 529.144,Z 1180.21,A -85,B 0,C 180,E1 25093.986,E2 25093.986} C_VEL
LIN {X 0,Y 529.991,Z 1172.231,A -85,B 0,C 180,E1 25091.618,E2 25091.618} C_VEL
LIN {X 0,Y 531.113,Z 1163.147,A -85,B 0,C 180,E1 25089.273,E2 25089.273} C_VEL
LIN {X 0,Y 532.956,Z 1150.578,A -85,B 0,C 180,E1 25086.447,E2 25086.447} C_VEL
LIN {X 0,Y 535.175,Z 1136.993,A -85,B 0,C 180,E1 25083.838,E2 25083.838} C_VEL
LIN {X 0,Y 537.465,Z 1124.122,A -85,B 0,C 180,E1 25081.638,E2 25081.638} C_VEL
LIN {X 0,Y 540.141,Z 1110.288,A -85,B 0,C 180,E1 25079.522,E2 25079.522} C_VEL
LIN {X 0,Y 543.857,Z 1091.905,A -85,B 0,C 180,E1 25077.031,E2 25077.031} C_VEL
LIN {X 0,Y 547.229,Z 1074.009,A -85,B 0,C 180,E1 25074.99,E2 25074.99} C_VEL
LIN {X 0,Y 550.38,Z 1057.476,A -85,B 0,C 180,E1 25073.296,E2 25073.296} C_VEL
LIN {X 0,Y 553.619,Z 1040.456,A -85,B 0,C 180,E1 25071.723,E2 25071.723} C_VEL
LIN {X 0,Y 557.421,Z 1020.234,A -85,B 0,C 180,E1 25070.048,E2 25070.048} C_VEL
LIN {X 0,Y 561.868,Z 995.648,A -85,B 0,C 180,E1 25068.276,E2 25068.276} C_VEL
LIN {X 0,Y 565.289,Z 975.529,A -85,B 0,C 180,E1 25067.011,E2 25067.011} C_VEL
LIN {X 0,Y 568.425,Z 955.89,A -85,B 0,C 180,E1 25065.919,E2 25065.919} C_VEL
LIN {X 0,Y 571.574,Z 934.769,A -85,B 0,C 180,E1 25064.89,E2 25064.89} C_VEL
LIN {X 0,Y 575.088,Z 909.015,A -85,B 0,C 180,E1 25063.82,E2 25063.82} C_VEL
LIN {X 0,Y 578.032,Z 883.077,A -85,B 0,C 180,E1 25062.954,E2 25062.954} C_VEL
LIN {X 0,Y 580.147,Z 861.334,A -85,B 0,C 180,E1 25062.361,E2 25062.361} C_VEL
LIN {X 0,Y 581.896,Z 839.759,A -85,B 0,C 180,E1 25061.893,E2 25061.893} C_VEL
LIN {X 0,Y 583.33,Z 814.286,A -85,B 0,C 180,E1 25061.466,E2 25061.466} C_VEL
LIN {X 0,Y 590.287,Z 591.564,A -85,B 0,C 180,E1 25058.284,E2 25058.284} C_VEL
LIN {X 0,Y 596.051,Z 414.48,A -85,B 0,C 180,E1 25055.702,E2 25055.702} C_VEL
LIN {X 0,Y 580.712,Z 392.107,A -85,B 0,C 180,E1 25053.465,E2 25053.465} C_VEL
LIN {X 0,Y 563.408,Z 367.788,A -85,B 0,C 180,E1 25050.679,E2 25050.679} C_VEL
LIN {X 0,Y 550.836,Z 351.309,A -85,B 0,C 180,E1 25048.487,E2 25048.487} C_VEL
LIN {X 0,Y 548.921,Z 348.252,A -85,B 0,C 180,E1 25048.032,E2 25048.032} C_VEL
LIN {X 0,Y 543.051,Z 337.478,A -85,B 0,C 180,E1 25045.873,E2 25045.873} C_VEL
LIN {X 0,Y 540.357,Z 332.678,A -85,B 0,C 180,E1 25044.838,E2 25044.838} C_VEL
LIN {X 0,Y 537.737,Z 328.001,A -85,B 0,C 180,E1 25043.797,E2 25043.797} C_VEL
LIN {X 0,Y 534.961,Z 323.047,A -85,B 0,C 180,E1 25042.646,E2 25042.646} C_VEL
LIN {X 0,Y 532.921,Z 319.418,A -85,B 0,C 180,E1 25041.766,E2 25041.766} C_VEL
LIN {X 0,Y 531.732,Z 317.619,A -85,B 0,C 180,E1 25041.28,E2 25041.28} C_VEL
LIN {X 0,Y 529.903,Z 314.358,A -85,B 0,C 180,E1 25040.431,E2 25040.431} C_VEL
LIN {X 0,Y 529.696,Z 313.329,A -85,B 0,C 180,E1 25040.094,E2 25040.094} C_VEL
LIN {X 0,Y 529.666,Z 313.18,A -85,B 0,C 180,E1 25036.675,E2 25036.675} C_VEL
LIN {X 0,Y 529.675,Z 313.239,A -85,B 0,C 180,E1 25033.315,E2 25033.315} C_VEL
LIN {X 0,Y 529.673,Z 313.168,A -85,B 0,C 180,E1 25029.812,E2 25029.812} C_VEL
LIN {X 0,Y 529.669,Z 313.253,A -85,B 0,C 180,E1 25026.395,E2 25026.395} C_VEL
LIN {X 0,Y 529.682,Z 313.252,A -85,B 0,C 180,E1 25022.922,E2 25022.922} C_VEL
LIN {X 0,Y 529.689,Z 313.25,A -85,B 0,C 180,E1 25019.459,E2 25019.459} C_VEL
LIN {X 0,Y 529.662,Z 313.254,A -85,B 0,C 180,E1 25015.995,E2 25015.995} C_VEL
LIN {X 0,Y 529.688,Z 313.247,A -85,B 0,C 180,E1 25012.516,E2 25012.516} C_VEL
LIN {X 0,Y 529.685,Z 313.247,A -85,B 0,C 180,E1 25008.984,E2 25008.984} C_VEL
LIN {X 0,Y 529.659,Z 313.248,A -85,B 0,C 180,E1 25005.56,E2 25005.56} C_VEL
LIN {X 0,Y 529.67,Z 313.245,A -85,B 0,C 180,E1 25002.064,E2 25002.064} C_VEL
LIN {X 0,Y 529.69,Z 313.243,A -85,B 0,C 180,E1 24998.634,E2 24998.634} C_VEL
LIN {X 0,Y 529.647,Z 313.176,A -85,B 0,C 180,E1 24995.233,E2 24995.233} C_VEL
LIN {X 0,Y 529.658,Z 313.255,A -85,B 0,C 180,E1 24991.716,E2 24991.716} C_VEL
LIN {X 0,Y 529.682,Z 313.174,A -85,B 0,C 180,E1 24988.346,E2 24988.346} C_VEL
LIN {X 0,Y 529.692,Z 313.521,A -85,B 0,C 180,E1 24985.577,E2 24985.577} C_VEL
LIN {X 0,Y 531.159,Z 316.968,A -85,B 0,C 180,E1 24984.696,E2 24984.696} C_VEL
LIN {X 0,Y 532.554,Z 318.785,A -85,B 0,C 180,E1 24984.141,E2 24984.141} C_VEL
LIN {X 0,Y 534.443,Z 322.576,A -85,B 0,C 180,E1 24983.224,E2 24983.224} C_VEL
LIN {X 0,Y 535.512,Z 324.327,A -85,B 0,C 180,E1 24982.774,E2 24982.774} C_VEL
LIN {X 0,Y 538.298,Z 329.73,A -85,B 0,C 180,E1 24981.518,E2 24981.518} C_VEL
LIN {X 0,Y 540.973,Z 334.751,A -85,B 0,C 180,E1 24980.381,E2 24980.381} C_VEL
LIN {X 0,Y 545.433,Z 343.288,A -85,B 0,C 180,E1 24978.563,E2 24978.563} C_VEL
LIN {X 0,Y 547.881,Z 347.941,A -85,B 0,C 180,E1 24977.667,E2 24977.667} C_VEL
LIN {X 0,Y 559.699,Z 363.777,A -85,B 0,C 180,E1 24975.549,E2 24975.549} C_VEL
LIN {X 0,Y 571.857,Z 380.687,A -85,B 0,C 180,E1 24973.551,E2 24973.551} C_VEL
LIN {X 0,Y 587.061,Z 403.049,A -85,B 0,C 180,E1 24971.228,E2 24971.228} C_VEL
LIN {X 0,Y 590.58,Z 408.562,A -85,B 0,C 180,E1 24970.716,E2 24970.716} C_VEL
LIN {X 0,Y 582.869,Z 637.199,A -85,B 0,C 180,E1 24967.461,E2 24967.461} C_VEL
LIN {X 0,Y 581.324,Z 684.43,A -85,B 0,C 180,E1 24966.792,E2 24966.792} C_VEL
LIN {X 0,Y 580.402,Z 692.129,A -85,B 0,C 180,E1 24966.753,E2 24966.753} C_VEL
LIN {X 0,Y 575.394,Z 712.72,A -85,B 0,C 180,E1 24966.914,E2 24966.914} C_VEL
LIN {X 0,Y 574.65,Z 719.328,A -85,B 0,C 180,E1 24966.875,E2 24966.875} C_VEL
LIN {X 0,Y 572.185,Z 787.358,A -85,B 0,C 180,E1 24965.888,E2 24965.888} C_VEL
LIN {X 0,Y 570.22,Z 815.453,A -85,B 0,C 180,E1 24965.313,E2 24965.313} C_VEL
LIN {X 0,Y 568.124,Z 837.573,A -85,B 0,C 180,E1 24964.704,E2 24964.704} C_VEL
LIN {X 0,Y 565.487,Z 860.87,A -85,B 0,C 180,E1 24963.907,E2 24963.907} C_VEL
LIN {X 0,Y 562.11,Z 885.615,A -85,B 0,C 180,E1 24962.855,E2 24962.855} C_VEL
LIN {X 0,Y 558.997,Z 905.62,A -85,B 0,C 180,E1 24961.847,E2 24961.847} C_VEL
LIN {X 0,Y 555.481,Z 926.361,A -85,B 0,C 180,E1 24960.636,E2 24960.636} C_VEL
LIN {X 0,Y 551.272,Z 948.982,A -85,B 0,C 180,E1 24959.083,E2 24959.083} C_VEL
LIN {X 0,Y 547.831,Z 966.221,A -85,B 0,C 180,E1 24957.722,E2 24957.722} C_VEL
LIN {X 0,Y 544.326,Z 983.129,A -85,B 0,C 180,E1 24956.217,E2 24956.217} C_VEL
LIN {X 0,Y 540.243,Z 1002.479,A -85,B 0,C 180,E1 24954.259,E2 24954.259} C_VEL
LIN {X 0,Y 536.437,Z 1019.724,A -85,B 0,C 180,E1 24952.233,E2 24952.233} C_VEL
LIN {X 0,Y 533.285,Z 1034.309,A -85,B 0,C 180,E1 24950.295,E2 24950.295} C_VEL
LIN {X 0,Y 529.869,Z 1050.773,A -85,B 0,C 180,E1 24947.8,E2 24947.8} C_VEL
LIN {X 0,Y 527.232,Z 1063.832,A -85,B 0,C 180,E1 24945.509,E2 24945.509} C_VEL
LIN {X 0,Y 525.236,Z 1074.862,A -85,B 0,C 180,E1 24943.317,E2 24943.317} C_VEL
LIN {X 0,Y 523.27,Z 1086.869,A -85,B 0,C 180,E1 24940.57,E2 24940.57} C_VEL
LIN {X 0,Y 521.947,Z 1096.181,A -85,B 0,C 180,E1 24938.039,E2 24938.039} C_VEL
LIN {X 0,Y 521.072,Z 1103.803,A -85,B 0,C 180,E1 24935.616,E2 24935.616} C_VEL
LIN {X 0,Y 520.405,Z 1111.455,A -85,B 0,C 180,E1 24932.643,E2 24932.643} C_VEL
LIN {X 0,Y 520.09,Z 1116.513,A -85,B 0,C 180,E1 24930.11,E2 24930.11} C_VEL
LIN {X 0,Y 519.949,Z 1120.952,A -85,B 0,C 180,E1 24927.244,E2 24927.244} C_VEL
LIN {X 0,Y 519.9,Z 1123.731,A -85,B 0,C 180,E1 24924.371,E2 24924.371} C_VEL
LIN {X 0,Y 519.917,Z 1124.783,A -85,B 0,C 180,E1 24922.041,E2 24922.041} C_VEL
LIN {X 0,Y 519.9,Z 1124.771,A -85,B 0,C 180,E1 24919.809,E2 24919.809} C_VEL
LIN {X 0,Y 519.918,Z 1123.608,A -85,B 0,C 180,E1 24917.336,E2 24917.336} C_VEL
LIN {X 0,Y 519.962,Z 1120.551,A -85,B 0,C 180,E1 24914.383,E2 24914.383} C_VEL
LIN {X 0,Y 520.114,Z 1116.203,A -85,B 0,C 180,E1 24911.623,E2 24911.623} C_VEL
LIN {X 0,Y 520.488,Z 1110.536,A -85,B 0,C 180,E1 24908.829,E2 24908.829} C_VEL
LIN {X 0,Y 521.143,Z 1103.353,A -85,B 0,C 180,E1 24906.12,E2 24906.12} C_VEL
LIN {X 0,Y 522.066,Z 1095.637,A -85,B 0,C 180,E1 24903.682,E2 24903.682} C_VEL
LIN {X 0,Y 523.619,Z 1085.084,A -85,B 0,C 180,E1 24900.861,E2 24900.861} C_VEL
LIN {X 0,Y 525.506,Z 1073.784,A -85,B 0,C 180,E1 24898.323,E2 24898.323} C_VEL
LIN {X 0,Y 527.721,Z 1062.086,A -85,B 0,C 180,E1 24896.018,E2 24896.018} C_VEL
LIN {X 0,Y 530.928,Z 1046.373,A -85,B 0,C 180,E1 24893.346,E2 24893.346} C_VEL
LIN {X 0,Y 533.928,Z 1032.448,A -85,B 0,C 180,E1 24891.284,E2 24891.284} C_VEL
LIN {X 0,Y 537.665,Z 1015.902,A -85,B 0,C 180,E1 24889.111,E2 24889.111} C_VEL
LIN {X 0,Y 541.774,Z 997.332,A -85,B 0,C 180,E1 24887.006,E2 24887.006} C_VEL
LIN {X 0,Y 545.495,Z 980.585,A -85,B 0,C 180,E1 24885.333,E2 24885.333} C_VEL
LIN {X 0,Y 550.045,Z 959.747,A -85,B 0,C 180,E1 24883.507,E2 24883.507} C_VEL
LIN {X 0,Y 554.179,Z 939.422,A -85,B 0,C 180,E1 24881.984,E2 24881.984} C_VEL
LIN {X 0,Y 557.745,Z 920.846,A -85,B 0,C 180,E1 24880.764,E2 24880.764} C_VEL
LIN {X 0,Y 561.74,Z 898.695,A -85,B 0,C 180,E1 24879.502,E2 24879.502} C_VEL
LIN {X 0,Y 565.303,Z 875.786,A -85,B 0,C 180,E1 24878.414,E2 24878.414} C_VEL
LIN {X 0,Y 568.034,Z 855.964,A -85,B 0,C 180,E1 24877.618,E2 24877.618} C_VEL
LIN {X 0,Y 570.605,Z 834.364,A -85,B 0,C 180,E1 24876.894,E2 24876.894} C_VEL
LIN {X 0,Y 573.225,Z 806.936,A -85,B 0,C 180,E1 24876.181,E2 24876.181} C_VEL
LIN {X 0,Y 574.754,Z 784.177,A -85,B 0,C 180,E1 24875.748,E2 24875.748} C_VEL
LIN {X 0,Y 584.102,Z 550.766,A -85,B 0,C 180,E1 24872.336,E2 24872.336} C_VEL
LIN {X 0,Y 589.84,Z 413.775,A -85,B 0,C 180,E1 24870.314,E2 24870.314} C_VEL
LIN {X 0,Y 580.307,Z 399.083,A -85,B 0,C 180,E1 24868.564,E2 24868.564} C_VEL
LIN {X 0,Y 570.644,Z 385.454,A -85,B 0,C 180,E1 24866.652,E2 24866.652} C_VEL
LIN {X 0,Y 561.43,Z 372.999,A -85,B 0,C 180,E1 24864.658,E2 24864.658} C_VEL
LIN {X 0,Y 555.914,Z 366.091,A -85,B 0,C 180,E1 24863.366,E2 24863.366} C_VEL
LIN {X 0,Y 551.973,Z 361.082,A -85,B 0,C 180,E1 24862.387,E2 24862.387} C_VEL
LIN {X 0,Y 544.239,Z 351.568,A -85,B 0,C 180,E1 24860.318,E2 24860.318} C_VEL
LIN {X 0,Y 540.81,Z 347.095,A -85,B 0,C 180,E1 24859.214,E2 24859.214} C_VEL
LIN {X 0,Y 537.907,Z 341.617,A -85,B 0,C 180,E1 24857.414,E2 24857.414} C_VEL
LIN {X 0,Y 535.244,Z 337.174,A -85,B 0,C 180,E1 24855.716,E2 24855.716} C_VEL
LIN {X 0,Y 534.264,Z 335.571,A -85,B 0,C 180,E1 24855.055,E2 24855.055} C_VEL
LIN {X 0,Y 532.182,Z 331.823,A -85,B 0,C 180,E1 24853.473,E2 24853.473} C_VEL
LIN {X 0,Y 530.868,Z 329.953,A -85,B 0,C 180,E1 24852.51,E2 24852.51} C_VEL
LIN {X 0,Y 528.781,Z 325.832,A -85,B 0,C 180,E1 24850.5,E2 24850.5} C_VEL
LIN {X 0,Y 525.61,Z 321.128,A -85,B 0,C 180,E1 24847.213,E2 24847.213} C_VEL
LIN {X 0,Y 524.876,Z 319.704,A -85,B 0,C 180,E1 24846.124,E2 24846.124} C_VEL
LIN {X 0,Y 522.117,Z 315.8,A -85,B 0,C 180,E1 24840.439,E2 24840.439} C_VEL
LIN {X 0,Y 521.941,Z 315.257,A -85,B 0,C 180,E1 24837.255,E2 24837.255} C_VEL
LIN {X 0,Y 522.329,Z 316.394,A -85,B 0,C 180,E1 24834.067,E2 24834.067} C_VEL
LIN {X 0,Y 525.407,Z 320.294,A -85,B 0,C 180,E1 24828.918,E2 24828.918} C_VEL
LIN {X 0,Y 527.876,Z 324.774,A -85,B 0,C 180,E1 24825.968,E2 24825.968} C_VEL
LIN {X 0,Y 529.078,Z 326.319,A -85,B 0,C 180,E1 24824.949,E2 24824.949} C_VEL
LIN {X 0,Y 531.412,Z 330.465,A -85,B 0,C 180,E1 24822.931,E2 24822.931} C_VEL
LIN {X 0,Y 532.567,Z 332.009,A -85,B 0,C 180,E1 24822.149,E2 24822.149} C_VEL
LIN {X 0,Y 534.787,Z 335.914,A -85,B 0,C 180,E1 24820.561,E2 24820.561} C_VEL
LIN {X 0,Y 535.838,Z 337.449,A -85,B 0,C 180,E1 24819.919,E2 24819.919} C_VEL
LIN {X 0,Y 538.036,Z 341.347,A -85,B 0,C 180,E1 24818.524,E2 24818.524} C_VEL
LIN {X 0,Y 538.969,Z 342.84,A -85,B 0,C 180,E1 24817.991,E2 24817.991} C_VEL
LIN {X 0,Y 541.496,Z 347.002,A -85,B 0,C 180,E1 24816.609,E2 24816.609} C_VEL
LIN {X 0,Y 543.519,Z 350.531,A -85,B 0,C 180,E1 24815.722,E2 24815.722} C_VEL
LIN {X 0,Y 547.065,Z 354.747,A -85,B 0,C 180,E1 24814.737,E2 24814.737} C_VEL
LIN {X 0,Y 551.396,Z 360.044,A -85,B 0,C 180,E1 24813.594,E2 24813.594} C_VEL
LIN {X 0,Y 555.523,Z 365.122,A -85,B 0,C 180,E1 24812.563,E2 24812.563} C_VEL
LIN {X 0,Y 563.244,Z 375.02,A -85,B 0,C 180,E1 24810.778,E2 24810.778} C_VEL
LIN {X 0,Y 571.641,Z 386.391,A -85,B 0,C 180,E1 24808.988,E2 24808.988} C_VEL
LIN {X 0,Y 581.857,Z 400.923,A -85,B 0,C 180,E1 24806.992,E2 24806.992} C_VEL
LIN {X 0,Y 592.588,Z 418.052,A -85,B 0,C 180,E1 24805.065,E2 24805.065} C_VEL
LIN {X 0,Y 593.001,Z 419.173,A -85,B 0,C 180,E1 24804.985,E2 24804.985} C_VEL
LIN {X 0,Y 584.663,Z 627.208,A -85,B 0,C 180,E1 24801.863,E2 24801.863} C_VEL
LIN {X 0,Y 577.405,Z 822.952,A -85,B 0,C 180,E1 24798.973,E2 24798.973} C_VEL
LIN {X 0,Y 575.463,Z 850.24,A -85,B 0,C 180,E1 24798.463,E2 24798.463} C_VEL
LIN {X 0,Y 572.762,Z 876.949,A -85,B 0,C 180,E1 24797.772,E2 24797.772} C_VEL
LIN {X 0,Y 570.261,Z 898.158,A -85,B 0,C 180,E1 24797.093,E2 24797.093} C_VEL
LIN {X 0,Y 567.484,Z 919.153,A -85,B 0,C 180,E1 24796.294,E2 24796.294} C_VEL
LIN {X 0,Y 564.167,Z 941.881,A -85,B 0,C 180,E1 24795.282,E2 24795.282} C_VEL
LIN {X 0,Y 559.823,Z 968.727,A -85,B 0,C 180,E1 24793.866,E2 24793.866} C_VEL
LIN {X 0,Y 556.354,Z 988.667,A -85,B 0,C 180,E1 24792.651,E2 24792.651} C_VEL
LIN {X 0,Y 552.803,Z 1008.147,A -85,B 0,C 180,E1 24791.313,E2 24791.313} C_VEL
LIN {X 0,Y 549.225,Z 1027.108,A -85,B 0,C 180,E1 24789.852,E2 24789.852} C_VEL
LIN {X 0,Y 544.927,Z 1049.468,A -85,B 0,C 180,E1 24787.907,E2 24787.907} C_VEL
LIN {X 0,Y 540.862,Z 1069.755,A -85,B 0,C 180,E1 24785.875,E2 24785.875} C_VEL
LIN {X 0,Y 537.619,Z 1086.134,A -85,B 0,C 180,E1 24784.042,E2 24784.042} C_VEL
LIN {X 0,Y 534.514,Z 1102.018,A -85,B 0,C 180,E1 24782.069,E2 24782.069} C_VEL
LIN {X 0,Y 532.421,Z 1112.597,A -85,B 0,C 180,E1 24780.592,E2 24780.592} C_VEL
LIN {X 0,Y 529.767,Z 1125.767,A -85,B 0,C 180,E1 24778.522,E2 24778.522} C_VEL
LIN {X 0,Y 526.998,Z 1140.795,A -85,B 0,C 180,E1 24775.873,E2 24775.873} C_VEL
LIN {X 0,Y 524.687,Z 1154.224,A -85,B 0,C 180,E1 24773.114,E2 24773.114} C_VEL
LIN {X 0,Y 523.153,Z 1164.517,A -85,B 0,C 180,E1 24770.706,E2 24770.706} C_VEL
LIN {X 0,Y 521.994,Z 1173.509,A -85,B 0,C 180,E1 24768.309,E2 24768.309} C_VEL
LIN {X 0,Y 521.012,Z 1183.011,A -85,B 0,C 180,E1 24765.357,E2 24765.357} C_VEL
LIN {X 0,Y 520.406,Z 1190.307,A -85,B 0,C 180,E1 24762.539,E2 24762.539} C_VEL
LIN {X 0,Y 520.13,Z 1195.489,A -85,B 0,C 180,E1 24760.075,E2 24760.075} C_VEL
LIN {X 0,Y 519.985,Z 1199.52,A -85,B 0,C 180,E1 24757.624,E2 24757.624} C_VEL
LIN {X 0,Y 519.929,Z 1202.43,A -85,B 0,C 180,E1 24755.186,E2 24755.186} C_VEL
LIN {X 0,Y 519.908,Z 1204.439,A -85,B 0,C 180,E1 24752.425,E2 24752.425} C_VEL
LIN {X 0,Y 519.895,Z 1204.894,A -85,B 0,C 180,E1 24749.449,E2 24749.449} C_VEL
LIN {X 0,Y 519.916,Z 1204.035,A -85,B 0,C 180,E1 24746.913,E2 24746.913} C_VEL
LIN {X 0,Y 519.934,Z 1202.088,A -85,B 0,C 180,E1 24744.482,E2 24744.482} C_VEL
LIN {X 0,Y 520.006,Z 1198.981,A -85,B 0,C 180,E1 24742.001,E2 24742.001} C_VEL
LIN {X 0,Y 520.194,Z 1194.113,A -85,B 0,C 180,E1 24739.181,E2 24739.181} C_VEL
LIN {X 0,Y 520.666,Z 1186.969,A -85,B 0,C 180,E1 24736.111,E2 24736.111} C_VEL
LIN {X 0,Y 521.282,Z 1179.856,A -85,B 0,C 180,E1 24733.623,E2 24733.623} C_VEL
LIN {X 0,Y 522.187,Z 1171.889,A -85,B 0,C 180,E1 24731.236,E2 24731.236} C_VEL
LIN {X 0,Y 523.471,Z 1162.229,A -85,B 0,C 180,E1 24728.721,E2 24728.721} C_VEL
LIN {X 0,Y 525.624,Z 1148.532,A -85,B 0,C 180,E1 24725.672,E2 24725.672} C_VEL
LIN {X 0,Y 527.756,Z 1136.356,A -85,B 0,C 180,E1 24723.32,E2 24723.32} C_VEL
LIN {X 0,Y 530.042,Z 1124.368,A -85,B 0,C 180,E1 24721.248,E2 24721.248} C_VEL
LIN {X 0,Y 532.758,Z 1111.056,A -85,B 0,C 180,E1 24719.179,E2 24719.179} C_VEL
LIN {X 0,Y 534.935,Z 1099.93,A -85,B 0,C 180,E1 24717.658,E2 24717.658} C_VEL
LIN {X 0,Y 538.035,Z 1084.298,A -85,B 0,C 180,E1 24715.731,E2 24715.731} C_VEL
LIN {X 0,Y 542.042,Z 1064.484,A -85,B 0,C 180,E1 24713.541,E2 24713.541} C_VEL
LIN {X 0,Y 546.189,Z 1043.312,A -85,B 0,C 180,E1 24711.508,E2 24711.508} C_VEL
LIN {X 0,Y 549.817,Z 1024.812,A -85,B 0,C 180,E1 24709.927,E2 24709.927} C_VEL
LIN {X 0,Y 553.455,Z 1005.727,A -85,B 0,C 180,E1 24708.47,E2 24708.47} C_VEL
LIN {X 0,Y 557.937,Z 981.403,A -85,B 0,C 180,E1 24706.836,E2 24706.836} C_VEL
LIN {X 0,Y 561.898,Z 957.775,A -85,B 0,C 180,E1 24705.485,E2 24705.485} C_VEL
LIN {X 0,Y 565.13,Z 937.023,A -85,B 0,C 180,E1 24704.455,E2 24704.455} C_VEL
LIN {X 0,Y 568.103,Z 916.146,A -85,B 0,C 180,E1 24703.558,E2 24703.558} C_VEL
LIN {X 0,Y 571.371,Z 890.525,A -85,B 0,C 180,E1 24702.629,E2 24702.629} C_VEL
LIN {X 0,Y 574.15,Z 863.577,A -85,B 0,C 180,E1 24701.863,E2 24701.863} C_VEL
LIN {X 0,Y 576.022,Z 841.663,A -85,B 0,C 180,E1 24701.374,E2 24701.374} C_VEL
LIN {X 0,Y 577.411,Z 819.262,A -85,B 0,C 180,E1 24700.985,E2 24700.985} C_VEL
LIN {X 0,Y 584.427,Z 605.058,A -85,B 0,C 180,E1 24697.9,E2 24697.9} C_VEL
LIN {X 0,Y 590.777,Z 418.443,A -85,B 0,C 180,E1 24695.17,E2 24695.17} C_VEL
LIN {X 0,Y 575.075,Z 395.596,A -85,B 0,C 180,E1 24692.823,E2 24692.823} C_VEL
LIN {X 0,Y 559.663,Z 373.817,A -85,B 0,C 180,E1 24690.283,E2 24690.283} C_VEL
LIN {X 0,Y 547.717,Z 357.971,A -85,B 0,C 180,E1 24688.158,E2 24688.158} C_VEL
LIN {X 0,Y 540.969,Z 348.803,A -85,B 0,C 180,E1 24686.808,E2 24686.808} C_VEL
LIN {X 0,Y 535.519,Z 338.96,A -85,B 0,C 180,E1 24684.724,E2 24684.724} C_VEL
LIN {X 0,Y 532.625,Z 333.899,A -85,B 0,C 180,E1 24683.57,E2 24683.57} C_VEL
LIN {X 0,Y 530.163,Z 329.338,A -85,B 0,C 180,E1 24682.511,E2 24682.511} C_VEL
LIN {X 0,Y 528.003,Z 325.419,A -85,B 0,C 180,E1 24681.554,E2 24681.554} C_VEL
LIN {X 0,Y 525.109,Z 320.646,A -85,B 0,C 180,E1 24680.277,E2 24680.277} C_VEL
LIN {X 0,Y 524.197,Z 319.066,A -85,B 0,C 180,E1 24679.848,E2 24679.848} C_VEL
LIN {X 0,Y 522.094,Z 315.793,A -85,B 0,C 180,E1 24678.885,E2 24678.885} C_VEL
LIN {X 0,Y 521.755,Z 314.376,A -85,B 0,C 180,E1 24678.453,E2 24678.453} C_VEL
LIN {X 0,Y 521.74,Z 314.166,A -85,B 0,C 180,E1 24674.994,E2 24674.994} C_VEL
LIN {X 0,Y 521.736,Z 314.194,A -85,B 0,C 180,E1 24671.609,E2 24671.609} C_VEL
LIN {X 0,Y 521.724,Z 314.175,A -85,B 0,C 180,E1 24668.153,E2 24668.153} C_VEL
LIN {X 0,Y 521.739,Z 314.221,A -85,B 0,C 180,E1 24664.727,E2 24664.727} C_VEL
LIN {X 0,Y 521.741,Z 314.22,A -85,B 0,C 180,E1 24661.208,E2 24661.208} C_VEL
LIN {X 0,Y 521.725,Z 314.221,A -85,B 0,C 180,E1 24657.803,E2 24657.803} C_VEL
LIN {X 0,Y 521.73,Z 314.222,A -85,B 0,C 180,E1 24654.281,E2 24654.281} C_VEL
LIN {X 0,Y 521.745,Z 314.223,A -85,B 0,C 180,E1 24650.847,E2 24650.847} C_VEL
LIN {X 0,Y 521.73,Z 314.226,A -85,B 0,C 180,E1 24647.38,E2 24647.38} C_VEL
LIN {X 0,Y 521.724,Z 314.227,A -85,B 0,C 180,E1 24643.98,E2 24643.98} C_VEL
LIN {X 0,Y 521.747,Z 314.226,A -85,B 0,C 180,E1 24640.521,E2 24640.521} C_VEL
LIN {X 0,Y 521.725,Z 314.213,A -85,B 0,C 180,E1 24637.104,E2 24637.104} C_VEL
LIN {X 0,Y 521.708,Z 314.172,A -85,B 0,C 180,E1 24633.599,E2 24633.599} C_VEL
LIN {X 0,Y 521.746,Z 314.188,A -85,B 0,C 180,E1 24630.24,E2 24630.24} C_VEL
LIN {X 0,Y 521.736,Z 314.431,A -85,B 0,C 180,E1 24627.264,E2 24627.264} C_VEL
LIN {X 0,Y 523.411,Z 318.192,A -85,B 0,C 180,E1 24626.198,E2 24626.198} C_VEL
LIN {X 0,Y 524.759,Z 320.176,A -85,B 0,C 180,E1 24625.591,E2 24625.591} C_VEL
LIN {X 0,Y 526.728,Z 323.784,A -85,B 0,C 180,E1 24624.621,E2 24624.621} C_VEL
LIN {X 0,Y 527.715,Z 325.494,A -85,B 0,C 180,E1 24624.163,E2 24624.163} C_VEL
LIN {X 0,Y 530.02,Z 329.417,A -85,B 0,C 180,E1 24623.136,E2 24623.136} C_VEL
LIN {X 0,Y 535.614,Z 340.336,A -85,B 0,C 180,E1 24620.601,E2 24620.601} C_VEL
LIN {X 0,Y 539.848,Z 348.03,A -85,B 0,C 180,E1 24618.959,E2 24618.959} C_VEL
LIN {X 0,Y 555.168,Z 368.514,A -85,B 0,C 180,E1 24616.099,E2 24616.099} C_VEL
LIN {X 0,Y 568.34,Z 387.064,A -85,B 0,C 180,E1 24613.885,E2 24613.885} C_VEL
LIN {X 0,Y 583.298,Z 409.245,A -85,B 0,C 180,E1 24611.561,E2 24611.561} C_VEL
LIN {X 0,Y 585.295,Z 412.59,A -85,B 0,C 180,E1 24611.26,E2 24611.26} C_VEL
LIN {X 0,Y 577.326,Z 640.171,A -85,B 0,C 180,E1 24608.001,E2 24608.001} C_VEL
LIN {X 0,Y 574.65,Z 719.328,A -85,B 0,C 180,E1 24606.875,E2 24606.875} C_VEL
LIN {X 0,Y 573.705,Z 727.027,A -85,B 0,C 180,E1 24606.839,E2 24606.839} C_VEL
LIN {X 0,Y 568.69,Z 747.613,A -85,B 0,C 180,E1 24607.002,E2 24607.002} C_VEL
LIN {X 0,Y 567.944,Z 754.22,A -85,B 0,C 180,E1 24606.963,E2 24606.963} C_VEL
LIN {X 0,Y 566.321,Z 793.174,A -85,B 0,C 180,E1 24606.37,E2 24606.37} C_VEL
LIN {X 0,Y 564.375,Z 817.859,A -85,B 0,C 180,E1 24605.832,E2 24605.832} C_VEL
LIN {X 0,Y 562.235,Z 839.45,A -85,B 0,C 180,E1 24605.226,E2 24605.226} C_VEL
LIN {X 0,Y 559.249,Z 864.751,A -85,B 0,C 180,E1 24604.338,E2 24604.338} C_VEL
LIN {X 0,Y 555.912,Z 887.817,A -85,B 0,C 180,E1 24603.33,E2 24603.33} C_VEL
LIN {X 0,Y 552.702,Z 907.647,A -85,B 0,C 180,E1 24602.315,E2 24602.315} C_VEL
LIN {X 0,Y 548.618,Z 930.828,A -85,B 0,C 180,E1 24600.927,E2 24600.927} C_VEL
LIN {X 0,Y 544.573,Z 951.351,A -85,B 0,C 180,E1 24599.476,E2 24599.476} C_VEL
LIN {X 0,Y 540.93,Z 968.917,A -85,B 0,C 180,E1 24598.061,E2 24598.061} C_VEL
LIN {X 0,Y 536.719,Z 988.615,A -85,B 0,C 180,E1 24596.26,E2 24596.26} C_VEL
LIN {X 0,Y 532.492,Z 1007.189,A -85,B 0,C 180,E1 24594.281,E2 24594.281} C_VEL
LIN {X 0,Y 529.04,Z 1022.402,A -85,B 0,C 180,E1 24592.443,E2 24592.443} C_VEL
LIN {X 0,Y 525.334,Z 1039.148,A -85,B 0,C 180,E1 24590.151,E2 24590.151} C_VEL
LIN {X 0,Y 521.964,Z 1054.276,A -85,B 0,C 180,E1 24587.733,E2 24587.733} C_VEL
LIN {X 0,Y 519.539,Z 1065.897,A -85,B 0,C 180,E1 24585.63,E2 24585.63} C_VEL
LIN {X 0,Y 517.095,Z 1078.897,A -85,B 0,C 180,E1 24582.948,E2 24582.948} C_VEL
LIN {X 0,Y 515.282,Z 1089.371,A -85,B 0,C 180,E1 24580.396,E2 24580.396} C_VEL
LIN {X 0,Y 514.061,Z 1097.717,A -85,B 0,C 180,E1 24578.05,E2 24578.05} C_VEL
LIN {X 0,Y 513.049,Z 1106.37,A -85,B 0,C 180,E1 24575.188,E2 24575.188} C_VEL
LIN {X 0,Y 512.43,Z 1112.891,A -85,B 0,C 180,E1 24572.46,E2 24572.46} C_VEL
LIN {X 0,Y 512.136,Z 1117.409,A -85,B 0,C 180,E1 24570.112,E2 24570.112} C_VEL
LIN {X 0,Y 511.986,Z 1121.2,A -85,B 0,C 180,E1 24567.538,E2 24567.538} C_VEL
LIN {X 0,Y 511.911,Z 1124.016,A -85,B 0,C 180,E1 24564.508,E2 24564.508} C_VEL
LIN {X 0,Y 511.921,Z 1125.051,A -85,B 0,C 180,E1 24562.029,E2 24562.029} C_VEL
LIN {X 0,Y 511.906,Z 1125.01,A -85,B 0,C 180,E1 24559.648,E2 24559.648} C_VEL
LIN {X 0,Y 511.929,Z 1123.662,A -85,B 0,C 180,E1 24556.79,E2 24556.79} C_VEL
LIN {X 0,Y 511.991,Z 1120.741,A -85,B 0,C 180,E1 24554.017,E2 24554.017} C_VEL
LIN {X 0,Y 512.157,Z 1117.237,A -85,B 0,C 180,E1 24551.681,E2 24551.681} C_VEL
LIN {X 0,Y 512.492,Z 1112.177,A -85,B 0,C 180,E1 24549.082,E2 24549.082} C_VEL
LIN {X 0,Y 513.267,Z 1104.44,A -85,B 0,C 180,E1 24546.016,E2 24546.016} C_VEL
LIN {X 0,Y 514.233,Z 1096.859,A -85,B 0,C 180,E1 24543.56,E2 24543.56} C_VEL
LIN {X 0,Y 515.833,Z 1086.716,A -85,B 0,C 180,E1 24540.76,E2 24540.76} C_VEL
LIN {X 0,Y 517.902,Z 1074.981,A -85,B 0,C 180,E1 24538.063,E2 24538.063} C_VEL
LIN {X 0,Y 520.092,Z 1063.995,A -85,B 0,C 180,E1 24535.85,E2 24535.85} C_VEL
LIN {X 0,Y 523.278,Z 1049.367,A -85,B 0,C 180,E1 24533.268,E2 24533.268} C_VEL
LIN {X 0,Y 526.755,Z 1033.949,A -85,B 0,C 180,E1 24530.929,E2 24530.929} C_VEL
LIN {X 0,Y 530.188,Z 1019.372,A -85,B 0,C 180,E1 24528.97,E2 24528.97} C_VEL
LIN {X 0,Y 534.849,Z 999.63,A -85,B 0,C 180,E1 24526.655,E2 24526.655} C_VEL
LIN {X 0,Y 538.788,Z 982.701,A -85,B 0,C 180,E1 24524.93,E2 24524.93} C_VEL
LIN {X 0,Y 542.864,Z 964.846,A -85,B 0,C 180,E1 24523.321,E2 24523.321} C_VEL
LIN {X 0,Y 547.797,Z 942.078,A -85,B 0,C 180,E1 24521.553,E2 24521.553} C_VEL
LIN {X 0,Y 551.664,Z 922.842,A -85,B 0,C 180,E1 24520.267,E2 24520.267} C_VEL
LIN {X 0,Y 555.383,Z 902.946,A -85,B 0,C 180,E1 24519.11,E2 24519.11} C_VEL
LIN {X 0,Y 559.588,Z 877.813,A -85,B 0,C 180,E1 24517.879,E2 24517.879} C_VEL
LIN {X 0,Y 562.618,Z 856.72,A -85,B 0,C 180,E1 24517.024,E2 24517.024} C_VEL
LIN {X 0,Y 565.289,Z 835.062,A -85,B 0,C 180,E1 24516.293,E2 24516.293} C_VEL
LIN {X 0,Y 568.013,Z 807.615,A -85,B 0,C 180,E1 24515.575,E2 24515.575} C_VEL
LIN {X 0,Y 569.603,Z 784.831,A -85,B 0,C 180,E1 24515.139,E2 24515.139} C_VEL
LIN {X 0,Y 579.357,Z 551.499,A -85,B 0,C 180,E1 24511.706,E2 24511.706} C_VEL
LIN {X 0,Y 585.213,Z 418.003,A -85,B 0,C 180,E1 24509.731,E2 24509.731} C_VEL
LIN {X 0,Y 576.085,Z 403.974,A -85,B 0,C 180,E1 24508.002,E2 24508.002} C_VEL
LIN {X 0,Y 565.44,Z 388.749,A -85,B 0,C 180,E1 24505.814,E2 24505.814} C_VEL
LIN {X 0,Y 554.74,Z 374.571,A -85,B 0,C 180,E1 24503.362,E2 24503.362} C_VEL
LIN {X 0,Y 548.914,Z 367.32,A -85,B 0,C 180,E1 24501.899,E2 24501.899} C_VEL
LIN {X 0,Y 542.218,Z 358.925,A -85,B 0,C 180,E1 24500.06,E2 24500.06} C_VEL
LIN {X 0,Y 537.262,Z 353.022,A -85,B 0,C 180,E1 24498.557,E2 24498.557} C_VEL
LIN {X 0,Y 533.505,Z 348.297,A -85,B 0,C 180,E1 24497.309,E2 24497.309} C_VEL
LIN {X 0,Y 530.605,Z 343.435,A -85,B 0,C 180,E1 24495.521,E2 24495.521} C_VEL
LIN {X 0,Y 527.703,Z 338.403,A -85,B 0,C 180,E1 24493.366,E2 24493.366} C_VEL
LIN {X 0,Y 526.254,Z 336.356,A -85,B 0,C 180,E1 24492.287,E2 24492.287} C_VEL
LIN {X 0,Y 523.956,Z 331.977,A -85,B 0,C 180,E1 24490.044,E2 24490.044} C_VEL
LIN {X 0,Y 521.272,Z 327.708,A -85,B 0,C 180,E1 24487.052,E2 24487.052} C_VEL
LIN {X 0,Y 520.523,Z 326.376,A -85,B 0,C 180,E1 24485.954,E2 24485.954} C_VEL
LIN {X 0,Y 517.972,Z 322.649,A -85,B 0,C 180,E1 24480.442,E2 24480.442} C_VEL
LIN {X 0,Y 517.784,Z 322.096,A -85,B 0,C 180,E1 24477.233,E2 24477.233} C_VEL
LIN {X 0,Y 518.22,Z 323.29,A -85,B 0,C 180,E1 24474.019,E2 24474.019} C_VEL
LIN {X 0,Y 521.255,Z 327.169,A -85,B 0,C 180,E1 24468.941,E2 24468.941} C_VEL
LIN {X 0,Y 523.73,Z 331.628,A -85,B 0,C 180,E1 24465.968,E2 24465.968} C_VEL
LIN {X 0,Y 524.852,Z 333.189,A -85,B 0,C 180,E1 24464.983,E2 24464.983} C_VEL
LIN {X 0,Y 527.137,Z 337.187,A -85,B 0,C 180,E1 24463.015,E2 24463.015} C_VEL
LIN {X 0,Y 528.231,Z 338.688,A -85,B 0,C 180,E1 24462.256,E2 24462.256} C_VEL
LIN {X 0,Y 530.486,Z 342.632,A -85,B 0,C 180,E1 24460.626,E2 24460.626} C_VEL
LIN {X 0,Y 531.485,Z 344.252,A -85,B 0,C 180,E1 24459.977,E2 24459.977} C_VEL
LIN {X 0,Y 533.932,Z 348.304,A -85,B 0,C 180,E1 24458.466,E2 24458.466} C_VEL
LIN {X 0,Y 538.15,Z 353.781,A -85,B 0,C 180,E1 24456.976,E2 24456.976} C_VEL
LIN {X 0,Y 544.917,Z 362.008,A -85,B 0,C 180,E1 24455.008,E2 24455.008} C_VEL
LIN {X 0,Y 549.289,Z 367.435,A -85,B 0,C 180,E1 24453.834,E2 24453.834} C_VEL
LIN {X 0,Y 553.275,Z 372.415,A -85,B 0,C 180,E1 24452.821,E2 24452.821} C_VEL
LIN {X 0,Y 560.688,Z 382.043,A -85,B 0,C 180,E1 24451.071,E2 24451.071} C_VEL
LIN {X 0,Y 570.852,Z 395.879,A -85,B 0,C 180,E1 24448.888,E2 24448.888} C_VEL
LIN {X 0,Y 580.826,Z 410.776,A -85,B 0,C 180,E1 24446.926,E2 24446.926} C_VEL
LIN {X 0,Y 588.247,Z 423.012,A -85,B 0,C 180,E1 24445.567,E2 24445.567} C_VEL
LIN {X 0,Y 579.51,Z 631.189,A -85,B 0,C 180,E1 24442.422,E2 24442.422} C_VEL
LIN {X 0,Y 572.049,Z 822.759,A -85,B 0,C 180,E1 24439.572,E2 24439.572} C_VEL
LIN {X 0,Y 569.984,Z 850.344,A -85,B 0,C 180,E1 24439.05,E2 24439.05} C_VEL
LIN {X 0,Y 567.21,Z 876.573,A -85,B 0,C 180,E1 24438.367,E2 24438.367} C_VEL
LIN {X 0,Y 564.58,Z 897.898,A -85,B 0,C 180,E1 24437.679,E2 24437.679} C_VEL
LIN {X 0,Y 561.662,Z 918.91,A -85,B 0,C 180,E1 24436.873,E2 24436.873} C_VEL
LIN {X 0,Y 558.229,Z 941.299,A -85,B 0,C 180,E1 24435.869,E2 24435.869} C_VEL
LIN {X 0,Y 553.763,Z 967.613,A -85,B 0,C 180,E1 24434.472,E2 24434.472} C_VEL
LIN {X 0,Y 549.813,Z 989.174,A -85,B 0,C 180,E1 24433.139,E2 24433.139} C_VEL
LIN {X 0,Y 545.977,Z 1009.261,A -85,B 0,C 180,E1 24431.735,E2 24431.735} C_VEL
LIN {X 0,Y 541.487,Z 1032.255,A -85,B 0,C 180,E1 24429.916,E2 24429.916} C_VEL
LIN {X 0,Y 536.972,Z 1054.078,A -85,B 0,C 180,E1 24427.913,E2 24427.913} C_VEL
LIN {X 0,Y 533.488,Z 1070.893,A -85,B 0,C 180,E1 24426.183,E2 24426.183} C_VEL
LIN {X 0,Y 530.067,Z 1087.477,A -85,B 0,C 180,E1 24424.287,E2 24424.287} C_VEL
LIN {X 0,Y 526.268,Z 1106.365,A -85,B 0,C 180,E1 24421.866,E2 24421.866} C_VEL
LIN {X 0,Y 523.006,Z 1122.91,A -85,B 0,C 180,E1 24419.427,E2 24419.427} C_VEL
LIN {X 0,Y 520.523,Z 1135.079,A -85,B 0,C 180,E1 24417.328,E2 24417.328} C_VEL
LIN {X 0,Y 518.359,Z 1146.554,A -85,B 0,C 180,E1 24415.11,E2 24415.11} C_VEL
LIN {X 0,Y 516.429,Z 1157.826,A -85,B 0,C 180,E1 24412.661,E2 24412.661} C_VEL
LIN {X 0,Y 514.577,Z 1170.267,A -85,B 0,C 180,E1 24409.524,E2 24409.524} C_VEL
LIN {X 0,Y 513.512,Z 1178.798,A -85,B 0,C 180,E1 24406.982,E2 24406.982} C_VEL
LIN {X 0,Y 512.82,Z 1185.755,A -85,B 0,C 180,E1 24404.567,E2 24404.567} C_VEL
LIN {X 0,Y 512.357,Z 1191.693,A -85,B 0,C 180,E1 24402.114,E2 24402.114} C_VEL
LIN {X 0,Y 512.077,Z 1197.139,A -85,B 0,C 180,E1 24399.327,E2 24399.327} C_VEL
LIN {X 0,Y 511.947,Z 1201.478,A -85,B 0,C 180,E1 24396.206,E2 24396.206} C_VEL
LIN {X 0,Y 511.914,Z 1203.76,A -85,B 0,C 180,E1 24393.583,E2 24393.583} C_VEL
LIN {X 0,Y 511.914,Z 1204.758,A -85,B 0,C 180,E1 24391.231,E2 24391.231} C_VEL
LIN {X 0,Y 511.909,Z 1204.803,A -85,B 0,C 180,E1 24388.993,E2 24388.993} C_VEL
LIN {X 0,Y 511.916,Z 1203.896,A -85,B 0,C 180,E1 24386.641,E2 24386.641} C_VEL
LIN {X 0,Y 511.939,Z 1201.858,A -85,B 0,C 180,E1 24384.171,E2 24384.171} C_VEL
LIN {X 0,Y 512.032,Z 1198.398,A -85,B 0,C 180,E1 24381.465,E2 24381.465} C_VEL
LIN {X 0,Y 512.306,Z 1192.594,A -85,B 0,C 180,E1 24378.289,E2 24378.289} C_VEL
LIN {X 0,Y 512.768,Z 1186.36,A -85,B 0,C 180,E1 24375.662,E2 24375.662} C_VEL
LIN {X 0,Y 513.435,Z 1179.502,A -85,B 0,C 180,E1 24373.249,E2 24373.249} C_VEL
LIN {X 0,Y 514.411,Z 1171.483,A -85,B 0,C 180,E1 24370.823,E2 24370.823} C_VEL
LIN {X 0,Y 516.054,Z 1160.383,A -85,B 0,C 180,E1 24367.922,E2 24367.922} C_VEL
LIN {X 0,Y 518.201,Z 1147.487,A -85,B 0,C 180,E1 24365.079,E2 24365.079} C_VEL
LIN {X 0,Y 520.396,Z 1135.719,A -85,B 0,C 180,E1 24362.788,E2 24362.788} C_VEL
LIN {X 0,Y 522.853,Z 1123.636,A -85,B 0,C 180,E1 24360.689,E2 24360.689} C_VEL
LIN {X 0,Y 525.64,Z 1109.578,A -85,B 0,C 180,E1 24358.588,E2 24358.588} C_VEL
LIN {X 0,Y 529.644,Z 1089.819,A -85,B 0,C 180,E1 24355.973,E2 24355.973} C_VEL
LIN {X 0,Y 533.302,Z 1072.242,A -85,B 0,C 180,E1 24353.935,E2 24353.935} C_VEL
LIN {X 0,Y 536.777,Z 1055.64,A -85,B 0,C 180,E1 24352.206,E2 24352.206} C_VEL
LIN {X 0,Y 540.469,Z 1037.908,A -85,B 0,C 180,E1 24350.545,E2 24350.545} C_VEL
LIN {X 0,Y 545.09,Z 1015.393,A -85,B 0,C 180,E1 24348.674,E2 24348.674} C_VEL
LIN {X 0,Y 549.49,Z 992.509,A -85,B 0,C 180,E1 24347.036,E2 24347.036} C_VEL
LIN {X 0,Y 552.878,Z 974.107,A -85,B 0,C 180,E1 24345.873,E2 24345.873} C_VEL
LIN {X 0,Y 556.12,Z 955.26,A -85,B 0,C 180,E1 24344.814,E2 24344.814} C_VEL
LIN {X 0,Y 559.286,Z 935.401,A -85,B 0,C 180,E1 24343.834,E2 24343.834} C_VEL
LIN {X 0,Y 562.444,Z 913.777,A -85,B 0,C 180,E1 24342.911,E2 24342.911} C_VEL
LIN {X 0,Y 566.078,Z 885.307,A -85,B 0,C 180,E1 24341.911,E2 24341.911} C_VEL
LIN {X 0,Y 568.552,Z 861.675,A -85,B 0,C 180,E1 24341.254,E2 24341.254} C_VEL
LIN {X 0,Y 570.431,Z 840.184,A -85,B 0,C 180,E1 24340.781,E2 24340.781} C_VEL
LIN {X 0,Y 571.867,Z 816.931,A -85,B 0,C 180,E1 24340.381,E2 24340.381} C_VEL
LIN {X 0,Y 579.329,Z 597.148,A -85,B 0,C 180,E1 24337.198,E2 24337.198} C_VEL
LIN {X 0,Y 585.509,Z 422.416,A -85,B 0,C 180,E1 24334.628,E2 24334.628} C_VEL
LIN {X 0,Y 569.383,Z 398.855,A -85,B 0,C 180,E1 24332.147,E2 24332.147} C_VEL
LIN {X 0,Y 555.293,Z 378.985,A -85,B 0,C 180,E1 24329.771,E2 24329.771} C_VEL
LIN {X 0,Y 544.373,Z 364.317,A -85,B 0,C 180,E1 24327.78,E2 24327.78} C_VEL
LIN {X 0,Y 536.657,Z 354.265,A -85,B 0,C 180,E1 24326.264,E2 24326.264} C_VEL
LIN {X 0,Y 532.502,Z 348.699,A -85,B 0,C 180,E1 24325.348,E2 24325.348} C_VEL
LIN {X 0,Y 528.099,Z 340.561,A -85,B 0,C 180,E1 24323.547,E2 24323.547} C_VEL
LIN {X 0,Y 525.012,Z 335.184,A -85,B 0,C 180,E1 24322.247,E2 24322.247} C_VEL
LIN {X 0,Y 522.455,Z 330.533,A -85,B 0,C 180,E1 24321.088,E2 24321.088} C_VEL
LIN {X 0,Y 520.331,Z 326.939,A -85,B 0,C 180,E1 24320.119,E2 24320.119} C_VEL
LIN {X 0,Y 519.419,Z 325.371,A -85,B 0,C 180,E1 24319.687,E2 24319.687} C_VEL
LIN {X 0,Y 517.347,Z 322.063,A -85,B 0,C 180,E1 24318.713,E2 24318.713} C_VEL
LIN {X 0,Y 516.581,Z 320.39,A -85,B 0,C 180,E1 24318.274,E2 24318.274} C_VEL
LIN {X 0,Y 514.292,Z 317.117,A -85,B 0,C 180,E1 24317.189,E2 24317.189} C_VEL
LIN {X 0,Y 513.817,Z 315.364,A -85,B 0,C 180,E1 24316.681,E2 24316.681} C_VEL
LIN {X 0,Y 513.796,Z 315.206,A -85,B 0,C 180,E1 24313.39,E2 24313.39} C_VEL
LIN {X 0,Y 513.794,Z 315.141,A -85,B 0,C 180,E1 24309.861,E2 24309.861} C_VEL
LIN {X 0,Y 513.791,Z 315.231,A -85,B 0,C 180,E1 24306.369,E2 24306.369} C_VEL
LIN {X 0,Y 513.804,Z 315.23,A -85,B 0,C 180,E1 24302.9,E2 24302.9} C_VEL
LIN {X 0,Y 513.81,Z 315.23,A -85,B 0,C 180,E1 24299.331,E2 24299.331} C_VEL
LIN {X 0,Y 513.785,Z 315.233,A -85,B 0,C 180,E1 24295.871,E2 24295.871} C_VEL
LIN {X 0,Y 513.801,Z 315.228,A -85,B 0,C 180,E1 24292.396,E2 24292.396} C_VEL
LIN {X 0,Y 513.807,Z 315.226,A -85,B 0,C 180,E1 24288.892,E2 24288.892} C_VEL
LIN {X 0,Y 513.786,Z 315.225,A -85,B 0,C 180,E1 24285.46,E2 24285.46} C_VEL
LIN {X 0,Y 513.782,Z 315.227,A -85,B 0,C 180,E1 24281.857,E2 24281.857} C_VEL
LIN {X 0,Y 513.814,Z 315.224,A -85,B 0,C 180,E1 24278.42,E2 24278.42} C_VEL
LIN {X 0,Y 513.788,Z 315.144,A -85,B 0,C 180,E1 24274.896,E2 24274.896} C_VEL
LIN {X 0,Y 513.772,Z 315.229,A -85,B 0,C 180,E1 24271.395,E2 24271.395} C_VEL
LIN {X 0,Y 513.808,Z 315.439,A -85,B 0,C 180,E1 24269.053,E2 24269.053} C_VEL
LIN {X 0,Y 515.519,Z 319.214,A -85,B 0,C 180,E1 24267.897,E2 24267.897} C_VEL
LIN {X 0,Y 516.933,Z 321.288,A -85,B 0,C 180,E1 24267.207,E2 24267.207} C_VEL
LIN {X 0,Y 519.187,Z 325.237,A -85,B 0,C 180,E1 24266.047,E2 24266.047} C_VEL
LIN {X 0,Y 522.015,Z 330.252,A -85,B 0,C 180,E1 24264.657,E2 24264.657} C_VEL
LIN {X 0,Y 525.632,Z 337.132,A -85,B 0,C 180,E1 24262.913,E2 24262.913} C_VEL
LIN {X 0,Y 530.326,Z 346.063,A -85,B 0,C 180,E1 24260.794,E2 24260.794} C_VEL
LIN {X 0,Y 532.227,Z 349.055,A -85,B 0,C 180,E1 24260.231,E2 24260.231} C_VEL
LIN {X 0,Y 538.092,Z 356.655,A -85,B 0,C 180,E1 24259.043,E2 24259.043} C_VEL
LIN {X 0,Y 546.987,Z 368.385,A -85,B 0,C 180,E1 24257.333,E2 24257.333} C_VEL
LIN {X 0,Y 556.511,Z 381.603,A -85,B 0,C 180,E1 24255.623,E2 24255.623} C_VEL
LIN {X 0,Y 569.572,Z 400.356,A -85,B 0,C 180,E1 24253.456,E2 24253.456} C_VEL
LIN {X 0,Y 580.071,Z 416.425,A -85,B 0,C 180,E1 24251.816,E2 24251.816} C_VEL
LIN {X 0,Y 571.828,Z 642.83,A -85,B 0,C 180,E1 24248.555,E2 24248.555} C_VEL
LIN {X 0,Y 567.944,Z 754.22,A -85,B 0,C 180,E1 24246.963,E2 24246.963} C_VEL
LIN {X 0,Y 566.983,Z 761.919,A -85,B 0,C 180,E1 24246.929,E2 24246.929} C_VEL
LIN {X 0,Y 561.805,Z 782.474,A -85,B 0,C 180,E1 24247.083,E2 24247.083} C_VEL
LIN {X 0,Y 560.968,Z 789.061,A -85,B 0,C 180,E1 24247.03,E2 24247.03} C_VEL
LIN {X 0,Y 558.896,Z 816.538,A -85,B 0,C 180,E1 24246.457,E2 24246.457} C_VEL
LIN {X 0,Y 556.677,Z 838.57,A -85,B 0,C 180,E1 24245.845,E2 24245.845} C_VEL
LIN {X 0,Y 553.94,Z 861.324,A -85,B 0,C 180,E1 24245.06,E2 24245.06} C_VEL
LIN {X 0,Y 550.243,Z 886.772,A -85,B 0,C 180,E1 24243.97,E2 24243.97} C_VEL
LIN {X 0,Y 546.913,Z 906.823,A -85,B 0,C 180,E1 24242.948,E2 24242.948} C_VEL
LIN {X 0,Y 542.963,Z 928.614,A -85,B 0,C 180,E1 24241.656,E2 24241.656} C_VEL
LIN {X 0,Y 538.46,Z 950.935,A -85,B 0,C 180,E1 24240.09,E2 24240.09} C_VEL
LIN {X 0,Y 534.662,Z 968.625,A -85,B 0,C 180,E1 24238.664,E2 24238.664} C_VEL
LIN {X 0,Y 530.624,Z 986.756,A -85,B 0,C 180,E1 24237.008,E2 24237.008} C_VEL
LIN {X 0,Y 526.102,Z 1006.234,A -85,B 0,C 180,E1 24234.955,E2 24234.955} C_VEL
LIN {X 0,Y 522.446,Z 1021.618,A -85,B 0,C 180,E1 24233.099,E2 24233.099} C_VEL
LIN {X 0,Y 519.01,Z 1036.214,A -85,B 0,C 180,E1 24231.115,E2 24231.115} C_VEL
LIN {X 0,Y 515.093,Z 1053.258,A -85,B 0,C 180,E1 24228.445,E2 24228.445} C_VEL
LIN {X 0,Y 512.335,Z 1065.629,A -85,B 0,C 180,E1 24226.205,E2 24226.205} C_VEL
LIN {X 0,Y 509.993,Z 1077.128,A -85,B 0,C 180,E1 24223.838,E2 24223.838} C_VEL
LIN {X 0,Y 507.722,Z 1089.344,A -85,B 0,C 180,E1 24220.897,E2 24220.897} C_VEL
LIN {X 0,Y 506.37,Z 1097.763,A -85,B 0,C 180,E1 24218.516,E2 24218.516} C_VEL
LIN {X 0,Y 505.371,Z 1105.34,A -85,B 0,C 180,E1 24216.019,E2 24216.019} C_VEL
LIN {X 0,Y 504.585,Z 1112.915,A -85,B 0,C 180,E1 24212.953,E2 24212.953} C_VEL
LIN {X 0,Y 504.221,Z 1117.737,A -85,B 0,C 180,E1 24210.454,E2 24210.454} C_VEL
LIN {X 0,Y 504.047,Z 1121.297,A -85,B 0,C 180,E1 24208.067,E2 24208.067} C_VEL
LIN {X 0,Y 503.949,Z 1124.279,A -85,B 0,C 180,E1 24205.22,E2 24205.22} C_VEL
LIN {X 0,Y 503.936,Z 1125.648,A -85,B 0,C 180,E1 24202.361,E2 24202.361} C_VEL
LIN {X 0,Y 503.93,Z 1125.726,A -85,B 0,C 180,E1 24199.944,E2 24199.944} C_VEL
LIN {X 0,Y 503.956,Z 1124.751,A -85,B 0,C 180,E1 24197.468,E2 24197.468} C_VEL
LIN {X 0,Y 504.015,Z 1122.305,A -85,B 0,C 180,E1 24194.584,E2 24194.584} C_VEL
LIN {X 0,Y 504.201,Z 1118.27,A -85,B 0,C 180,E1 24191.74,E2 24191.74} C_VEL
LIN {X 0,Y 504.511,Z 1113.72,A -85,B 0,C 180,E1 24189.303,E2 24189.303} C_VEL
LIN {X 0,Y 505.242,Z 1106.902,A -85,B 0,C 180,E1 24186.391,E2 24186.391} C_VEL
LIN {X 0,Y 506.373,Z 1098.281,A -85,B 0,C 180,E1 24183.497,E2 24183.497} C_VEL
LIN {X 0,Y 507.682,Z 1090.091,A -85,B 0,C 180,E1 24181.15,E2 24181.15} C_VEL
LIN {X 0,Y 509.876,Z 1078.491,A -85,B 0,C 180,E1 24178.295,E2 24178.295} C_VEL
LIN {X 0,Y 512.328,Z 1066.554,A -85,B 0,C 180,E1 24175.802,E2 24175.802} C_VEL
LIN {X 0,Y 515.098,Z 1054.377,A -85,B 0,C 180,E1 24173.56,E2 24173.56} C_VEL
LIN {X 0,Y 518.997,Z 1038.029,A -85,B 0,C 180,E1 24170.934,E2 24170.934} C_VEL
LIN {X 0,Y 522.679,Z 1023.035,A -85,B 0,C 180,E1 24168.848,E2 24168.848} C_VEL
LIN {X 0,Y 526.435,Z 1008.012,A -85,B 0,C 180,E1 24166.992,E2 24166.992} C_VEL
LIN {X 0,Y 531.218,Z 988.739,A -85,B 0,C 180,E1 24164.898,E2 24164.898} C_VEL
LIN {X 0,Y 535.699,Z 969.865,A -85,B 0,C 180,E1 24163.132,E2 24163.132} C_VEL
LIN {X 0,Y 539.851,Z 951.852,A -85,B 0,C 180,E1 24161.649,E2 24161.649} C_VEL
LIN {X 0,Y 544.703,Z 929.504,A -85,B 0,C 180,E1 24160.053,E2 24160.053} C_VEL
LIN {X 0,Y 548.876,Z 908.288,A -85,B 0,C 180,E1 24158.77,E2 24158.77} C_VEL
LIN {X 0,Y 552.544,Z 887.909,A -85,B 0,C 180,E1 24157.709,E2 24157.709} C_VEL
LIN {X 0,Y 556.518,Z 862.948,A -85,B 0,C 180,E1 24156.62,E2 24156.62} C_VEL
LIN {X 0,Y 559.57,Z 839.66,A -85,B 0,C 180,E1 24155.801,E2 24155.801} C_VEL
LIN {X 0,Y 561.979,Z 817.737,A -85,B 0,C 180,E1 24155.18,E2 24155.18} C_VEL
LIN {X 0,Y 564.219,Z 790.959,A -85,B 0,C 180,E1 24154.608,E2 24154.608} C_VEL
LIN {X 0,Y 566.584,Z 739.59,A -85,B 0,C 180,E1 24153.828,E2 24153.828} C_VEL
LIN {X 0,Y 577.074,Z 499.225,A -85,B 0,C 180,E1 24150.279,E2 24150.279} C_VEL
LIN {X 0,Y 580.561,Z 422.097,A -85,B 0,C 180,E1 24149.12,E2 24149.12} C_VEL
LIN {X 0,Y 569.832,Z 405.685,A -85,B 0,C 180,E1 24147.003,E2 24147.003} C_VEL
LIN {X 0,Y 559.425,Z 391.105,A -85,B 0,C 180,E1 24144.752,E2 24144.752} C_VEL
LIN {X 0,Y 551.603,Z 380.792,A -85,B 0,C 180,E1 24142.881,E2 24142.881} C_VEL
LIN {X 0,Y 546.999,Z 374.893,A -85,B 0,C 180,E1 24141.697,E2 24141.697} C_VEL
LIN {X 0,Y 540.036,Z 366.104,A -85,B 0,C 180,E1 24139.749,E2 24139.749} C_VEL
LIN {X 0,Y 535.477,Z 360.551,A -85,B 0,C 180,E1 24138.339,E2 24138.339} C_VEL
LIN {X 0,Y 531.593,Z 355.649,A -85,B 0,C 180,E1 24137.035,E2 24137.035} C_VEL
LIN {X 0,Y 527.064,Z 350.577,A -85,B 0,C 180,E1 24135.402,E2 24135.402} C_VEL
LIN {X 0,Y 524.316,Z 347.428,A -85,B 0,C 180,E1 24134.241,E2 24134.241} C_VEL
LIN {X 0,Y 522.579,Z 343.809,A -85,B 0,C 180,E1 24132.711,E2 24132.711} C_VEL
LIN {X 0,Y 520.225,Z 339.885,A -85,B 0,C 180,E1 24130.633,E2 24130.633} C_VEL
LIN {X 0,Y 519.475,Z 338.539,A -85,B 0,C 180,E1 24129.864,E2 24129.864} C_VEL
LIN {X 0,Y 516.907,Z 334.121,A -85,B 0,C 180,E1 24126.777,E2 24126.777} C_VEL
LIN {X 0,Y 515.381,Z 332.239,A -85,B 0,C 180,E1 24124.674,E2 24124.674} C_VEL
LIN {X 0,Y 513.773,Z 329.336,A -85,B 0,C 180,E1 24120,E2 24120} C_VEL
LIN {X 0,Y 513.671,Z 328.997,A -85,B 0,C 180,E1 24116.916,E2 24116.916} C_VEL
LIN {X 0,Y 514.223,Z 330.402,A -85,B 0,C 180,E1 24113.637,E2 24113.637} C_VEL
LIN {X 0,Y 517.098,Z 334.053,A -85,B 0,C 180,E1 24108.964,E2 24108.964} C_VEL
LIN {X 0,Y 519.592,Z 338.488,A -85,B 0,C 180,E1 24105.967,E2 24105.967} C_VEL
LIN {X 0,Y 520.59,Z 339.907,A -85,B 0,C 180,E1 24105.086,E2 24105.086} C_VEL
LIN {X 0,Y 523.034,Z 344.088,A -85,B 0,C 180,E1 24102.993,E2 24102.993} C_VEL
LIN {X 0,Y 523.926,Z 345.452,A -85,B 0,C 180,E1 24102.335,E2 24102.335} C_VEL
LIN {X 0,Y 526.365,Z 349.456,A -85,B 0,C 180,E1 24100.699,E2 24100.699} C_VEL
LIN {X 0,Y 527.975,Z 351.477,A -85,B 0,C 180,E1 24100.069,E2 24100.069} C_VEL
LIN {X 0,Y 531.894,Z 355.824,A -85,B 0,C 180,E1 24098.669,E2 24098.669} C_VEL
LIN {X 0,Y 536.692,Z 361.636,A -85,B 0,C 180,E1 24097.084,E2 24097.084} C_VEL
LIN {X 0,Y 545.928,Z 373.055,A -85,B 0,C 180,E1 24094.419,E2 24094.419} C_VEL
LIN {X 0,Y 551.419,Z 380.228,A -85,B 0,C 180,E1 24092.984,E2 24092.984} C_VEL
LIN {X 0,Y 558.352,Z 389.35,A -85,B 0,C 180,E1 24091.319,E2 24091.319} C_VEL
LIN {X 0,Y 568.09,Z 402.785,A -85,B 0,C 180,E1 24089.19,E2 24089.19} C_VEL
LIN {X 0,Y 577.608,Z 417.194,A -85,B 0,C 180,E1 24087.276,E2 24087.276} C_VEL
LIN {X 0,Y 583.543,Z 427.111,A -85,B 0,C 180,E1 24086.155,E2 24086.155} C_VEL
LIN {X 0,Y 574.427,Z 635.615,A -85,B 0,C 180,E1 24082.988,E2 24082.988} C_VEL
LIN {X 0,Y 566.805,Z 822.071,A -85,B 0,C 180,E1 24080.191,E2 24080.191} C_VEL
LIN {X 0,Y 564.691,Z 849.472,A -85,B 0,C 180,E1 24079.673,E2 24079.673} C_VEL
LIN {X 0,Y 561.76,Z 876.14,A -85,B 0,C 180,E1 24078.978,E2 24078.978} C_VEL
LIN {X 0,Y 559.034,Z 897.411,A -85,B 0,C 180,E1 24078.29,E2 24078.29} C_VEL
LIN {X 0,Y 556.042,Z 918.01,A -85,B 0,C 180,E1 24077.498,E2 24077.498} C_VEL
LIN {X 0,Y 552.371,Z 940.902,A -85,B 0,C 180,E1 24076.465,E2 24076.465} C_VEL
LIN {X 0,Y 547.643,Z 967.444,A -85,B 0,C 180,E1 24075.042,E2 24075.042} C_VEL
LIN {X 0,Y 543.659,Z 988.15,A -85,B 0,C 180,E1 24073.75,E2 24073.75} C_VEL
LIN {X 0,Y 539.79,Z 1007.39,A -85,B 0,C 180,E1 24072.395,E2 24072.395} C_VEL
LIN {X 0,Y 535.486,Z 1028.328,A -85,B 0,C 180,E1 24070.737,E2 24070.737} C_VEL
LIN {X 0,Y 530.495,Z 1051.848,A -85,B 0,C 180,E1 24068.598,E2 24068.598} C_VEL
LIN {X 0,Y 526.829,Z 1068.82,A -85,B 0,C 180,E1 24066.851,E2 24066.851} C_VEL
LIN {X 0,Y 523.41,Z 1084.712,A -85,B 0,C 180,E1 24065.032,E2 24065.032} C_VEL
LIN {X 0,Y 520.058,Z 1100.399,A -85,B 0,C 180,E1 24063.041,E2 24063.041} C_VEL
LIN {X 0,Y 516.344,Z 1118.345,A -85,B 0,C 180,E1 24060.487,E2 24060.487} C_VEL
LIN {X 0,Y 513.201,Z 1134.214,A -85,B 0,C 180,E1 24057.878,E2 24057.878} C_VEL
LIN {X 0,Y 511.357,Z 1143.686,A -85,B 0,C 180,E1 24056.1,E2 24056.1} C_VEL
LIN {X 0,Y 509.183,Z 1155.25,A -85,B 0,C 180,E1 24053.615,E2 24053.615} C_VEL
LIN {X 0,Y 507.543,Z 1164.973,A -85,B 0,C 180,E1 24051.253,E2 24051.253} C_VEL
LIN {X 0,Y 506.26,Z 1173.912,A -85,B 0,C 180,E1 24048.779,E2 24048.779} C_VEL
LIN {X 0,Y 505.112,Z 1183.63,A -85,B 0,C 180,E1 24045.617,E2 24045.617} C_VEL
LIN {X 0,Y 504.469,Z 1190.63,A -85,B 0,C 180,E1 24042.792,E2 24042.792} C_VEL
LIN {X 0,Y 504.157,Z 1195.69,A -85,B 0,C 180,E1 24040.282,E2 24040.282} C_VEL
LIN {X 0,Y 504.002,Z 1199.515,A -85,B 0,C 180,E1 24037.868,E2 24037.868} C_VEL
LIN {X 0,Y 503.932,Z 1202.424,A -85,B 0,C 180,E1 24035.351,E2 24035.351} C_VEL
LIN {X 0,Y 503.91,Z 1204.438,A -85,B 0,C 180,E1 24032.502,E2 24032.502} C_VEL
LIN {X 0,Y 503.895,Z 1204.894,A -85,B 0,C 180,E1 24029.432,E2 24029.432} C_VEL
LIN {X 0,Y 503.916,Z 1204.029,A -85,B 0,C 180,E1 24026.815,E2 24026.815} C_VEL
LIN {X 0,Y 503.937,Z 1202.196,A -85,B 0,C 180,E1 24024.421,E2 24024.421} C_VEL
LIN {X 0,Y 504.008,Z 1199.354,A -85,B 0,C 180,E1 24022.018,E2 24022.018} C_VEL
LIN {X 0,Y 504.167,Z 1195.483,A -85,B 0,C 180,E1 24019.603,E2 24019.603} C_VEL
LIN {X 0,Y 504.523,Z 1190.047,A -85,B 0,C 180,E1 24016.943,E2 24016.943} C_VEL
LIN {X 0,Y 505.268,Z 1181.974,A -85,B 0,C 180,E1 24013.798,E2 24013.798} C_VEL
LIN {X 0,Y 506.326,Z 1173.402,A -85,B 0,C 180,E1 24011.073,E2 24011.073} C_VEL
LIN {X 0,Y 507.614,Z 1164.519,A -85,B 0,C 180,E1 24008.63,E2 24008.63} C_VEL
LIN {X 0,Y 509.278,Z 1154.743,A -85,B 0,C 180,E1 24006.267,E2 24006.267} C_VEL
LIN {X 0,Y 511.858,Z 1141.399,A -85,B 0,C 180,E1 24003.428,E2 24003.428} C_VEL
LIN {X 0,Y 514.691,Z 1126.547,A -85,B 0,C 180,E1 24000.817,E2 24000.817} C_VEL
LIN {X 0,Y 517.676,Z 1112.006,A -85,B 0,C 180,E1 23998.568,E2 23998.568} C_VEL
LIN {X 0,Y 520.728,Z 1097.569,A -85,B 0,C 180,E1 23996.559,E2 23996.559} C_VEL
LIN {X 0,Y 524.403,Z 1080.632,A -85,B 0,C 180,E1 23994.442,E2 23994.442} C_VEL
LIN {X 0,Y 529.159,Z 1058.772,A -85,B 0,C 180,E1 23992.045,E2 23992.045} C_VEL
LIN {X 0,Y 533.067,Z 1040.746,A -85,B 0,C 180,E1 23990.308,E2 23990.308} C_VEL
LIN {X 0,Y 536.884,Z 1022.791,A -85,B 0,C 180,E1 23988.756,E2 23988.756} C_VEL
LIN {X 0,Y 541.183,Z 1002.064,A -85,B 0,C 180,E1 23987.165,E2 23987.165} C_VEL
LIN {X 0,Y 546.145,Z 976.561,A -85,B 0,C 180,E1 23985.478,E2 23985.478} C_VEL
LIN {X 0,Y 549.756,Z 956.384,A -85,B 0,C 180,E1 23984.325,E2 23984.325} C_VEL
LIN {X 0,Y 553.105,Z 936.157,A -85,B 0,C 180,E1 23983.314,E2 23983.314} C_VEL
LIN {X 0,Y 556.263,Z 915.319,A -85,B 0,C 180,E1 23982.413,E2 23982.413} C_VEL
LIN {X 0,Y 559.781,Z 889.467,A -85,B 0,C 180,E1 23981.471,E2 23981.471} C_VEL
LIN {X 0,Y 562.741,Z 862.487,A -85,B 0,C 180,E1 23980.703,E2 23980.703} C_VEL
LIN {X 0,Y 564.719,Z 840.692,A -85,B 0,C 180,E1 23980.218,E2 23980.218} C_VEL
LIN {X 0,Y 566.186,Z 818.133,A -85,B 0,C 180,E1 23979.823,E2 23979.823} C_VEL
LIN {X 0,Y 573.76,Z 603.861,A -85,B 0,C 180,E1 23976.699,E2 23976.699} C_VEL
LIN {X 0,Y 580.254,Z 426.373,A -85,B 0,C 180,E1 23974.074,E2 23974.074} C_VEL
LIN {X 0,Y 564.531,Z 403.352,A -85,B 0,C 180,E1 23971.59,E2 23971.59} C_VEL
LIN {X 0,Y 551.6,Z 384.959,A -85,B 0,C 180,E1 23969.363,E2 23969.363} C_VEL
LIN {X 0,Y 539.045,Z 367.841,A -85,B 0,C 180,E1 23967,E2 23967} C_VEL
LIN {X 0,Y 528.637,Z 354.516,A -85,B 0,C 180,E1 23964.858,E2 23964.858} C_VEL
LIN {X 0,Y 524.232,Z 348.786,A -85,B 0,C 180,E1 23963.851,E2 23963.851} C_VEL
LIN {X 0,Y 520.246,Z 341.515,A -85,B 0,C 180,E1 23962.127,E2 23962.127} C_VEL
LIN {X 0,Y 517.383,Z 336.471,A -85,B 0,C 180,E1 23960.83,E2 23960.83} C_VEL
LIN {X 0,Y 514.643,Z 331.672,A -85,B 0,C 180,E1 23959.523,E2 23959.523} C_VEL
LIN {X 0,Y 512.441,Z 327.868,A -85,B 0,C 180,E1 23958.427,E2 23958.427} C_VEL
LIN {X 0,Y 511.309,Z 326.145,A -85,B 0,C 180,E1 23957.88,E2 23957.88} C_VEL
LIN {X 0,Y 509.292,Z 322.507,A -85,B 0,C 180,E1 23956.775,E2 23956.775} C_VEL
LIN {X 0,Y 508.23,Z 320.91,A -85,B 0,C 180,E1 23956.223,E2 23956.223} C_VEL
LIN {X 0,Y 506.231,Z 317.749,A -85,B 0,C 180,E1 23955.113,E2 23955.113} C_VEL
LIN {X 0,Y 505.881,Z 316.365,A -85,B 0,C 180,E1 23954.655,E2 23954.655} C_VEL
LIN {X 0,Y 505.854,Z 316.151,A -85,B 0,C 180,E1 23951.169,E2 23951.169} C_VEL
LIN {X 0,Y 505.864,Z 316.163,A -85,B 0,C 180,E1 23947.61,E2 23947.61} C_VEL
LIN {X 0,Y 505.848,Z 316.2,A -85,B 0,C 180,E1 23944.081,E2 23944.081} C_VEL
LIN {X 0,Y 505.864,Z 316.199,A -85,B 0,C 180,E1 23940.566,E2 23940.566} C_VEL
LIN {X 0,Y 505.863,Z 316.197,A -85,B 0,C 180,E1 23937.054,E2 23937.054} C_VEL
LIN {X 0,Y 505.855,Z 316.198,A -85,B 0,C 180,E1 23933.531,E2 23933.531} C_VEL
LIN {X 0,Y 505.843,Z 316.2,A -85,B 0,C 180,E1 23929.983,E2 23929.983} C_VEL
LIN {X 0,Y 505.868,Z 316.196,A -85,B 0,C 180,E1 23926.512,E2 23926.512} C_VEL
LIN {X 0,Y 505.864,Z 316.196,A -85,B 0,C 180,E1 23922.99,E2 23922.99} C_VEL
LIN {X 0,Y 505.837,Z 316.201,A -85,B 0,C 180,E1 23919.52,E2 23919.52} C_VEL
LIN {X 0,Y 505.853,Z 316.147,A -85,B 0,C 180,E1 23916.095,E2 23916.095} C_VEL
LIN {X 0,Y 505.868,Z 316.173,A -85,B 0,C 180,E1 23912.555,E2 23912.555} C_VEL
LIN {X 0,Y 505.91,Z 316.631,A -85,B 0,C 180,E1 23910.982,E2 23910.982} C_VEL
LIN {X 0,Y 507.707,Z 320.378,A -85,B 0,C 180,E1 23909.723,E2 23909.723} C_VEL
LIN {X 0,Y 509.055,Z 322.219,A -85,B 0,C 180,E1 23909.028,E2 23909.028} C_VEL
LIN {X 0,Y 511.086,Z 325.98,A -85,B 0,C 180,E1 23907.85,E2 23907.85} C_VEL
LIN {X 0,Y 512.171,Z 327.872,A -85,B 0,C 180,E1 23907.263,E2 23907.263} C_VEL
LIN {X 0,Y 514.957,Z 332.858,A -85,B 0,C 180,E1 23905.805,E2 23905.805} C_VEL
LIN {X 0,Y 517.695,Z 337.756,A -85,B 0,C 180,E1 23904.454,E2 23904.454} C_VEL
LIN {X 0,Y 520.816,Z 343.741,A -85,B 0,C 180,E1 23902.927,E2 23902.927} C_VEL
LIN {X 0,Y 523.011,Z 347.819,A -85,B 0,C 180,E1 23901.965,E2 23901.965} C_VEL
LIN {X 0,Y 534.439,Z 362.404,A -85,B 0,C 180,E1 23899.518,E2 23899.518} C_VEL
LIN {X 0,Y 545.731,Z 377.605,A -85,B 0,C 180,E1 23897.319,E2 23897.319} C_VEL
LIN {X 0,Y 557.886,Z 394.759,A -85,B 0,C 180,E1 23895.149,E2 23895.149} C_VEL
LIN {X 0,Y 572.111,Z 415.862,A -85,B 0,C 180,E1 23892.82,E2 23892.82} C_VEL
LIN {X 0,Y 574.895,Z 420.363,A -85,B 0,C 180,E1 23892.38,E2 23892.38} C_VEL
LIN {X 0,Y 566.32,Z 647.078,A -85,B 0,C 180,E1 23889.096,E2 23889.096} C_VEL
LIN {X 0,Y 561.109,Z 786.334,A -85,B 0,C 180,E1 23887.074,E2 23887.074} C_VEL
LIN {X 0,Y 560.968,Z 789.061,A -85,B 0,C 180,E1 23887.03,E2 23887.03} C_VEL
LIN {X 0,Y 559.568,Z 797.802,A -85,B 0,C 180,E1 23886.968,E2 23886.968} C_VEL
LIN {X 0,Y 554.352,Z 814.921,A -85,B 0,C 180,E1 23887.007,E2 23887.007} C_VEL
LIN {X 0,Y 552.829,Z 822.452,A -85,B 0,C 180,E1 23886.903,E2 23886.903} C_VEL
LIN {X 0,Y 552.717,Z 823.524,A -85,B 0,C 180,E1 23886.876,E2 23886.876} C_VEL
LIN {X 0,Y 549.882,Z 849.274,A -85,B 0,C 180,E1 23886.095,E2 23886.095} C_VEL
LIN {X 0,Y 546.962,Z 870.575,A -85,B 0,C 180,E1 23885.286,E2 23885.286} C_VEL
LIN {X 0,Y 543.779,Z 890.99,A -85,B 0,C 180,E1 23884.367,E2 23884.367} C_VEL
LIN {X 0,Y 540.046,Z 912.505,A -85,B 0,C 180,E1 23883.231,E2 23883.231} C_VEL
LIN {X 0,Y 535.512,Z 935.764,A -85,B 0,C 180,E1 23881.771,E2 23881.771} C_VEL
LIN {X 0,Y 531.668,Z 953.918,A -85,B 0,C 180,E1 23880.452,E2 23880.452} C_VEL
LIN {X 0,Y 527.767,Z 971.403,A -85,B 0,C 180,E1 23879.012,E2 23879.012} C_VEL
LIN {X 0,Y 522.842,Z 992.511,A -85,B 0,C 180,E1 23877.012,E2 23877.012} C_VEL
LIN {X 0,Y 518.812,Z 1009,A -85,B 0,C 180,E1 23875.208,E2 23875.208} C_VEL
LIN {X 0,Y 515.274,Z 1023.362,A -85,B 0,C 180,E1 23873.44,E2 23873.44} C_VEL
LIN {X 0,Y 511.158,Z 1040.306,A -85,B 0,C 180,E1 23871.08,E2 23871.08} C_VEL
LIN {X 0,Y 507.48,Z 1055.448,A -85,B 0,C 180,E1 23868.608,E2 23868.608} C_VEL
LIN {X 0,Y 504.78,Z 1067.089,A -85,B 0,C 180,E1 23866.454,E2 23866.454} C_VEL
LIN {X 0,Y 502.04,Z 1080.056,A -85,B 0,C 180,E1 23863.709,E2 23863.709} C_VEL
LIN {X 0,Y 499.879,Z 1091.006,A -85,B 0,C 180,E1 23860.954,E2 23860.954} C_VEL
LIN {X 0,Y 498.484,Z 1099.303,A -85,B 0,C 180,E1 23858.536,E2 23858.536} C_VEL
LIN {X 0,Y 497.302,Z 1107.98,A -85,B 0,C 180,E1 23855.538,E2 23855.538} C_VEL
LIN {X 0,Y 496.607,Z 1114.35,A -85,B 0,C 180,E1 23852.77,E2 23852.77} C_VEL
LIN {X 0,Y 496.26,Z 1118.833,A -85,B 0,C 180,E1 23850.346,E2 23850.346} C_VEL
LIN {X 0,Y 496.064,Z 1122.742,A -85,B 0,C 180,E1 23847.574,E2 23847.574} C_VEL
LIN {X 0,Y 495.971,Z 1125.356,A -85,B 0,C 180,E1 23844.563,E2 23844.563} C_VEL
LIN {X 0,Y 495.974,Z 1126.35,A -85,B 0,C 180,E1 23842.121,E2 23842.121} C_VEL
LIN {X 0,Y 495.96,Z 1126.358,A -85,B 0,C 180,E1 23839.781,E2 23839.781} C_VEL
LIN {X 0,Y 495.987,Z 1125.297,A -85,B 0,C 180,E1 23837.188,E2 23837.188} C_VEL
LIN {X 0,Y 496.072,Z 1122.475,A -85,B 0,C 180,E1 23834.091,E2 23834.091} C_VEL
LIN {X 0,Y 496.272,Z 1118.905,A -85,B 0,C 180,E1 23831.56,E2 23831.56} C_VEL
LIN {X 0,Y 496.612,Z 1114.395,A -85,B 0,C 180,E1 23829.105,E2 23829.105} C_VEL
LIN {X 0,Y 497.403,Z 1107.62,A -85,B 0,C 180,E1 23826.157,E2 23826.157} C_VEL
LIN {X 0,Y 498.573,Z 1099.309,A -85,B 0,C 180,E1 23823.306,E2 23823.306} C_VEL
LIN {X 0,Y 499.963,Z 1091.176,A -85,B 0,C 180,E1 23820.924,E2 23820.924} C_VEL
LIN {X 0,Y 502.163,Z 1080.249,A -85,B 0,C 180,E1 23818.154,E2 23818.154} C_VEL
LIN {X 0,Y 504.891,Z 1067.72,A -85,B 0,C 180,E1 23815.473,E2 23815.473} C_VEL
LIN {X 0,Y 507.756,Z 1055.776,A -85,B 0,C 180,E1 23813.228,E2 23813.228} C_VEL
LIN {X 0,Y 511.618,Z 1040.557,A -85,B 0,C 180,E1 23810.708,E2 23810.708} C_VEL
LIN {X 0,Y 515.692,Z 1024.69,A -85,B 0,C 180,E1 23808.455,E2 23808.455} C_VEL
LIN {X 0,Y 519.542,Z 1009.989,A -85,B 0,C 180,E1 23806.603,E2 23806.603} C_VEL
LIN {X 0,Y 524.142,Z 992.394,A -85,B 0,C 180,E1 23804.64,E2 23804.64} C_VEL
LIN {X 0,Y 529.19,Z 972.159,A -85,B 0,C 180,E1 23802.694,E2 23802.694} C_VEL
LIN {X 0,Y 533.496,Z 954.266,A -85,B 0,C 180,E1 23801.195,E2 23801.195} C_VEL
LIN {X 0,Y 538.029,Z 934.469,A -85,B 0,C 180,E1 23799.74,E2 23799.74} C_VEL
LIN {X 0,Y 542.799,Z 911.556,A -85,B 0,C 180,E1 23798.306,E2 23798.306} C_VEL
LIN {X 0,Y 546.493,Z 892.013,A -85,B 0,C 180,E1 23797.262,E2 23797.262} C_VEL
LIN {X 0,Y 549.88,Z 872.214,A -85,B 0,C 180,E1 23796.356,E2 23796.356} C_VEL
LIN {X 0,Y 553.229,Z 849.886,A -85,B 0,C 180,E1 23795.492,E2 23795.492} C_VEL
LIN {X 0,Y 556.302,Z 824.187,A -85,B 0,C 180,E1 23794.705,E2 23794.705} C_VEL
LIN {X 0,Y 558.233,Z 804.087,A -85,B 0,C 180,E1 23794.224,E2 23794.224} C_VEL
LIN {X 0,Y 559.757,Z 782.408,A -85,B 0,C 180,E1 23793.822,E2 23793.822} C_VEL
LIN {X 0,Y 570.535,Z 543.633,A -85,B 0,C 180,E1 23790.274,E2 23790.274} C_VEL
LIN {X 0,Y 576.052,Z 426.39,A -85,B 0,C 180,E1 23788.512,E2 23788.512} C_VEL
LIN {X 0,Y 566.187,Z 411.334,A -85,B 0,C 180,E1 23786.51,E2 23786.51} C_VEL
LIN {X 0,Y 556.696,Z 397.826,A -85,B 0,C 180,E1 23784.4,E2 23784.4} C_VEL
LIN {X 0,Y 549.08,Z 387.675,A -85,B 0,C 180,E1 23782.54,E2 23782.54} C_VEL
LIN {X 0,Y 544.362,Z 381.555,A -85,B 0,C 180,E1 23781.299,E2 23781.299} C_VEL
LIN {X 0,Y 537.703,Z 373.092,A -85,B 0,C 180,E1 23779.386,E2 23779.386} C_VEL
LIN {X 0,Y 533.539,Z 367.922,A -85,B 0,C 180,E1 23778.069,E2 23778.069} C_VEL
LIN {X 0,Y 528.895,Z 362.22,A -85,B 0,C 180,E1 23776.474,E2 23776.474} C_VEL
LIN {X 0,Y 525.005,Z 357.508,A -85,B 0,C 180,E1 23775.012,E2 23775.012} C_VEL
LIN {X 0,Y 520.062,Z 351.825,A -85,B 0,C 180,E1 23772.943,E2 23772.943} C_VEL
LIN {X 0,Y 516.155,Z 347.417,A -85,B 0,C 180,E1 23770.944,E2 23770.944} C_VEL
LIN {X 0,Y 515.321,Z 345.42,A -85,B 0,C 180,E1 23769.944,E2 23769.944} C_VEL
LIN {X 0,Y 512.723,Z 341.087,A -85,B 0,C 180,E1 23766.832,E2 23766.832} C_VEL
LIN {X 0,Y 511.984,Z 339.846,A -85,B 0,C 180,E1 23765.716,E2 23765.716} C_VEL
LIN {X 0,Y 509.677,Z 336.275,A -85,B 0,C 180,E1 23760.225,E2 23760.225} C_VEL
LIN {X 0,Y 509.539,Z 335.828,A -85,B 0,C 180,E1 23757.075,E2 23757.075} C_VEL
LIN {X 0,Y 510.045,Z 337.106,A -85,B 0,C 180,E1 23753.923,E2 23753.923} C_VEL
LIN {X 0,Y 512.891,Z 340.751,A -85,B 0,C 180,E1 23749.099,E2 23749.099} C_VEL
LIN {X 0,Y 515.346,Z 345.221,A -85,B 0,C 180,E1 23746.079,E2 23746.079} C_VEL
LIN {X 0,Y 516.346,Z 346.635,A -85,B 0,C 180,E1 23745.19,E2 23745.19} C_VEL
LIN {X 0,Y 518.05,Z 349.736,A -85,B 0,C 180,E1 23743.805,E2 23743.805} C_VEL
LIN {X 0,Y 520.874,Z 352.662,A -85,B 0,C 180,E1 23742.517,E2 23742.517} C_VEL
LIN {X 0,Y 525.24,Z 357.518,A -85,B 0,C 180,E1 23740.714,E2 23740.714} C_VEL
LIN {X 0,Y 529.56,Z 362.859,A -85,B 0,C 180,E1 23739.092,E2 23739.092} C_VEL
LIN {X 0,Y 531.263,Z 364.9,A -85,B 0,C 180,E1 23738.498,E2 23738.498} C_VEL
LIN {X 0,Y 536.51,Z 371.356,A -85,B 0,C 180,E1 23736.786,E2 23736.786} C_VEL
LIN {X 0,Y 543.941,Z 380.598,A -85,B 0,C 180,E1 23734.64,E2 23734.64} C_VEL
LIN {X 0,Y 549.286,Z 387.634,A -85,B 0,C 180,E1 23733.222,E2 23733.222} C_VEL
LIN {X 0,Y 556.316,Z 397.041,A -85,B 0,C 180,E1 23731.503,E2 23731.503} C_VEL
LIN {X 0,Y 565.557,Z 410.023,A -85,B 0,C 180,E1 23729.45,E2 23729.45} C_VEL
LIN {X 0,Y 574.727,Z 424.121,A -85,B 0,C 180,E1 23727.569,E2 23727.569} C_VEL
LIN {X 0,Y 578.913,Z 431.296,A -85,B 0,C 180,E1 23726.753,E2 23726.753} C_VEL
LIN {X 0,Y 569.399,Z 640.257,A -85,B 0,C 180,E1 23723.561,E2 23723.561} C_VEL
LIN {X 0,Y 561.625,Z 821.833,A -85,B 0,C 180,E1 23720.817,E2 23720.817} C_VEL
LIN {X 0,Y 559.403,Z 849.481,A -85,B 0,C 180,E1 23720.291,E2 23720.291} C_VEL
LIN {X 0,Y 556.423,Z 875.597,A -85,B 0,C 180,E1 23719.607,E2 23719.607} C_VEL
LIN {X 0,Y 553.55,Z 897.091,A -85,B 0,C 180,E1 23718.909,E2 23718.909} C_VEL
LIN {X 0,Y 550.395,Z 917.9,A -85,B 0,C 180,E1 23718.104,E2 23718.104} C_VEL
LIN {X 0,Y 546.491,Z 941.284,A -85,B 0,C 180,E1 23717.041,E2 23717.041} C_VEL
LIN {X 0,Y 541.537,Z 967.68,A -85,B 0,C 180,E1 23715.605,E2 23715.605} C_VEL
LIN {X 0,Y 537.423,Z 988.1,A -85,B 0,C 180,E1 23714.315,E2 23714.315} C_VEL
LIN {X 0,Y 533.235,Z 1007.972,A -85,B 0,C 180,E1 23712.895,E2 23712.895} C_VEL
LIN {X 0,Y 528.217,Z 1031.253,A -85,B 0,C 180,E1 23711.005,E2 23711.005} C_VEL
LIN {X 0,Y 523.406,Z 1052.606,A -85,B 0,C 180,E1 23709.002,E2 23709.002} C_VEL
LIN {X 0,Y 519.622,Z 1069.402,A -85,B 0,C 180,E1 23707.241,E2 23707.241} C_VEL
LIN {X 0,Y 516.08,Z 1085.203,A -85,B 0,C 180,E1 23705.4,E2 23705.4} C_VEL
LIN {X 0,Y 512.397,Z 1101.784,A -85,B 0,C 180,E1 23703.252,E2 23703.252} C_VEL
LIN {X 0,Y 508.351,Z 1120.446,A -85,B 0,C 180,E1 23700.494,E2 23700.494} C_VEL
LIN {X 0,Y 505.567,Z 1134.049,A -85,B 0,C 180,E1 23698.208,E2 23698.208} C_VEL
LIN {X 0,Y 503.2,Z 1146.226,A -85,B 0,C 180,E1 23695.922,E2 23695.922} C_VEL
LIN {X 0,Y 501.735,Z 1154.219,A -85,B 0,C 180,E1 23694.237,E2 23694.237} C_VEL
LIN {X 0,Y 499.96,Z 1164.054,A -85,B 0,C 180,E1 23691.838,E2 23691.838} C_VEL
LIN {X 0,Y 498.603,Z 1172.695,A -85,B 0,C 180,E1 23689.444,E2 23689.444} C_VEL
LIN {X 0,Y 497.545,Z 1180.562,A -85,B 0,C 180,E1 23686.941,E2 23686.941} C_VEL
LIN {X 0,Y 496.701,Z 1188.758,A -85,B 0,C 180,E1 23683.86,E2 23683.86} C_VEL
LIN {X 0,Y 496.207,Z 1195.067,A -85,B 0,C 180,E1 23680.801,E2 23680.801} C_VEL
LIN {X 0,Y 496.019,Z 1199.192,A -85,B 0,C 180,E1 23678.228,E2 23678.228} C_VEL
LIN {X 0,Y 495.94,Z 1202.08,A -85,B 0,C 180,E1 23675.786,E2 23675.786} C_VEL
LIN {X 0,Y 495.915,Z 1203.958,A -85,B 0,C 180,E1 23673.352,E2 23673.352} C_VEL
LIN {X 0,Y 495.906,Z 1204.826,A -85,B 0,C 180,E1 23670.924,E2 23670.924} C_VEL
LIN {X 0,Y 495.91,Z 1204.712,A -85,B 0,C 180,E1 23668.498,E2 23668.498} C_VEL
LIN {X 0,Y 495.919,Z 1203.413,A -85,B 0,C 180,E1 23665.722,E2 23665.722} C_VEL
LIN {X 0,Y 495.988,Z 1200.309,A -85,B 0,C 180,E1 23662.587,E2 23662.587} C_VEL
LIN {X 0,Y 496.144,Z 1196.306,A -85,B 0,C 180,E1 23659.902,E2 23659.902} C_VEL
LIN {X 0,Y 496.455,Z 1191.316,A -85,B 0,C 180,E1 23657.319,E2 23657.319} C_VEL
LIN {X 0,Y 497.003,Z 1185.444,A -85,B 0,C 180,E1 23654.839,E2 23654.839} C_VEL
LIN {X 0,Y 497.897,Z 1177.734,A -85,B 0,C 180,E1 23652.107,E2 23652.107} C_VEL
LIN {X 0,Y 499.522,Z 1166.783,A -85,B 0,C 180,E1 23648.875,E2 23648.875} C_VEL
LIN {X 0,Y 501.326,Z 1156.414,A -85,B 0,C 180,E1 23646.273,E2 23646.273} C_VEL
LIN {X 0,Y 502.876,Z 1148.066,A -85,B 0,C 180,E1 23644.44,E2 23644.44} C_VEL
LIN {X 0,Y 505.293,Z 1135.465,A -85,B 0,C 180,E1 23642.033,E2 23642.033} C_VEL
LIN {X 0,Y 507.91,Z 1122.809,A -85,B 0,C 180,E1 23639.869,E2 23639.869} C_VEL
LIN {X 0,Y 511.102,Z 1107.946,A -85,B 0,C 180,E1 23637.587,E2 23637.587} C_VEL
LIN {X 0,Y 515.694,Z 1087.531,A -85,B 0,C 180,E1 23634.842,E2 23634.842} C_VEL
LIN {X 0,Y 519.452,Z 1070.976,A -85,B 0,C 180,E1 23632.884,E2 23632.884} C_VEL
LIN {X 0,Y 523.244,Z 1054.351,A -85,B 0,C 180,E1 23631.118,E2 23631.118} C_VEL
LIN {X 0,Y 527.256,Z 1036.59,A -85,B 0,C 180,E1 23629.425,E2 23629.425} C_VEL
LIN {X 0,Y 532.25,Z 1013.966,A -85,B 0,C 180,E1 23627.52,E2 23627.52} C_VEL
LIN {X 0,Y 536.97,Z 991.005,A -85,B 0,C 180,E1 23625.861,E2 23625.861} C_VEL
LIN {X 0,Y 540.824,Z 971.414,A -85,B 0,C 180,E1 23624.621,E2 23624.621} C_VEL
LIN {X 0,Y 544.428,Z 951.839,A -85,B 0,C 180,E1 23623.529,E2 23623.529} C_VEL
LIN {X 0,Y 548.347,Z 928.557,A -85,B 0,C 180,E1 23622.398,E2 23622.398} C_VEL
LIN {X 0,Y 552.275,Z 901.895,A -85,B 0,C 180,E1 23621.33,E2 23621.33} C_VEL
LIN {X 0,Y 555.123,Z 879.648,A -85,B 0,C 180,E1 23620.598,E2 23620.598} C_VEL
LIN {X 0,Y 557.492,Z 858.034,A -85,B 0,C 180,E1 23620.015,E2 23620.015} C_VEL
LIN {X 0,Y 559.581,Z 834.695,A -85,B 0,C 180,E1 23619.517,E2 23619.517} C_VEL
LIN {X 0,Y 561.422,Z 798.527,A -85,B 0,C 180,E1 23618.94,E2 23618.94} C_VEL
LIN {X 0,Y 569.617,Z 573.604,A -85,B 0,C 180,E1 23615.647,E2 23615.647} C_VEL
LIN {X 0,Y 574.977,Z 430.244,A -85,B 0,C 180,E1 23613.499,E2 23613.499} C_VEL
LIN {X 0,Y 558.182,Z 405.465,A -85,B 0,C 180,E1 23610.759,E2 23610.759} C_VEL
LIN {X 0,Y 545.347,Z 387.327,A -85,B 0,C 180,E1 23608.471,E2 23608.471} C_VEL
LIN {X 0,Y 534.475,Z 372.64,A -85,B 0,C 180,E1 23606.35,E2 23606.35} C_VEL
LIN {X 0,Y 526.481,Z 362.159,A -85,B 0,C 180,E1 23604.667,E2 23604.667} C_VEL
LIN {X 0,Y 518.566,Z 352.353,A -85,B 0,C 180,E1 23602.893,E2 23602.893} C_VEL
LIN {X 0,Y 515.717,Z 348.149,A -85,B 0,C 180,E1 23602.095,E2 23602.095} C_VEL
LIN {X 0,Y 512.595,Z 342.74,A -85,B 0,C 180,E1 23600.675,E2 23600.675} C_VEL
LIN {X 0,Y 509.875,Z 337.965,A -85,B 0,C 180,E1 23599.355,E2 23599.355} C_VEL
LIN {X 0,Y 507.71,Z 334.137,A -85,B 0,C 180,E1 23598.248,E2 23598.248} C_VEL
LIN {X 0,Y 504.764,Z 329.2,A -85,B 0,C 180,E1 23596.692,E2 23596.692} C_VEL
LIN {X 0,Y 503.742,Z 327.477,A -85,B 0,C 180,E1 23596.122,E2 23596.122} C_VEL
LIN {X 0,Y 501.607,Z 324.005,A -85,B 0,C 180,E1 23594.901,E2 23594.901} C_VEL
LIN {X 0,Y 500.734,Z 322.36,A -85,B 0,C 180,E1 23594.336,E2 23594.336} C_VEL
LIN {X 0,Y 498.421,Z 319.14,A -85,B 0,C 180,E1 23592.984,E2 23592.984} C_VEL
LIN {X 0,Y 497.938,Z 317.357,A -85,B 0,C 180,E1 23592.29,E2 23592.29} C_VEL
LIN {X 0,Y 497.917,Z 317.117,A -85,B 0,C 180,E1 23588.895,E2 23588.895} C_VEL
LIN {X 0,Y 497.924,Z 317.191,A -85,B 0,C 180,E1 23585.416,E2 23585.416} C_VEL
LIN {X 0,Y 497.914,Z 317.192,A -85,B 0,C 180,E1 23581.841,E2 23581.841} C_VEL
LIN {X 0,Y 497.912,Z 317.191,A -85,B 0,C 180,E1 23578.274,E2 23578.274} C_VEL
LIN {X 0,Y 497.927,Z 317.19,A -85,B 0,C 180,E1 23574.7,E2 23574.7} C_VEL
LIN {X 0,Y 497.93,Z 317.19,A -85,B 0,C 180,E1 23571.096,E2 23571.096} C_VEL
LIN {X 0,Y 497.906,Z 317.194,A -85,B 0,C 180,E1 23567.592,E2 23567.592} C_VEL
LIN {X 0,Y 497.909,Z 317.193,A -85,B 0,C 180,E1 23564.031,E2 23564.031} C_VEL
LIN {X 0,Y 497.931,Z 317.191,A -85,B 0,C 180,E1 23560.528,E2 23560.528} C_VEL
LIN {X 0,Y 497.909,Z 317.167,A -85,B 0,C 180,E1 23557.071,E2 23557.071} C_VEL
LIN {X 0,Y 497.905,Z 317.241,A -85,B 0,C 180,E1 23553.589,E2 23553.589} C_VEL
LIN {X 0,Y 498.033,Z 317.926,A -85,B 0,C 180,E1 23553.145,E2 23553.145} C_VEL
LIN {X 0,Y 499.998,Z 321.682,A -85,B 0,C 180,E1 23551.709,E2 23551.709} C_VEL
LIN {X 0,Y 501.228,Z 323.348,A -85,B 0,C 180,E1 23551.003,E2 23551.003} C_VEL
LIN {X 0,Y 503.294,Z 327.113,A -85,B 0,C 180,E1 23549.694,E2 23549.694} C_VEL
LIN {X 0,Y 504.344,Z 328.759,A -85,B 0,C 180,E1 23549.104,E2 23549.104} C_VEL
LIN {X 0,Y 506.653,Z 332.734,A -85,B 0,C 180,E1 23547.802,E2 23547.802} C_VEL
LIN {X 0,Y 509.504,Z 337.835,A -85,B 0,C 180,E1 23546.263,E2 23546.263} C_VEL
LIN {X 0,Y 512.015,Z 342.509,A -85,B 0,C 180,E1 23544.96,E2 23544.96} C_VEL
LIN {X 0,Y 515.21,Z 348.198,A -85,B 0,C 180,E1 23543.499,E2 23543.499} C_VEL
LIN {X 0,Y 527.765,Z 364.295,A -85,B 0,C 180,E1 23540.638,E2 23540.638} C_VEL
LIN {X 0,Y 537.058,Z 376.622,A -85,B 0,C 180,E1 23538.735,E2 23538.735} C_VEL
LIN {X 0,Y 548.536,Z 392.548,A -85,B 0,C 180,E1 23536.554,E2 23536.554} C_VEL
LIN {X 0,Y 563.042,Z 413.852,A -85,B 0,C 180,E1 23534.045,E2 23534.045} C_VEL
LIN {X 0,Y 569.754,Z 424.366,A -85,B 0,C 180,E1 23532.953,E2 23532.953} C_VEL
LIN {X 0,Y 560.883,Z 650.331,A -85,B 0,C 180,E1 23529.661,E2 23529.661} C_VEL
LIN {X 0,Y 555.607,Z 786.585,A -85,B 0,C 180,E1 23527.671,E2 23527.671} C_VEL
LIN {X 0,Y 553.702,Z 813.05,A -85,B 0,C 180,E1 23527.147,E2 23527.147} C_VEL
LIN {X 0,Y 552.717,Z 823.524,A -85,B 0,C 180,E1 23526.876,E2 23526.876} C_VEL
LIN {X 0,Y 551.3,Z 831.082,A -85,B 0,C 180,E1 23526.746,E2 23526.746} C_VEL
LIN {X 0,Y 544.873,Z 850.243,A -85,B 0,C 180,E1 23526.598,E2 23526.598} C_VEL
LIN {X 0,Y 543.174,Z 857.409,A -85,B 0,C 180,E1 23526.414,E2 23526.414} C_VEL
LIN {X 0,Y 540.238,Z 877.641,A -85,B 0,C 180,E1 23525.596,E2 23525.596} C_VEL
LIN {X 0,Y 535.925,Z 903.109,A -85,B 0,C 180,E1 23524.358,E2 23524.358} C_VEL
LIN {X 0,Y 532.139,Z 922.938,A -85,B 0,C 180,E1 23523.21,E2 23523.21} C_VEL
LIN {X 0,Y 528.531,Z 940.4,A -85,B 0,C 180,E1 23522.054,E2 23522.054} C_VEL
LIN {X 0,Y 524.148,Z 960.281,A -85,B 0,C 180,E1 23520.555,E2 23520.555} C_VEL
LIN {X 0,Y 519.171,Z 981.176,A -85,B 0,C 180,E1 23518.718,E2 23518.718} C_VEL
LIN {X 0,Y 515.129,Z 997.503,A -85,B 0,C 180,E1 23517.075,E2 23517.075} C_VEL
LIN {X 0,Y 511.047,Z 1013.615,A -85,B 0,C 180,E1 23515.246,E2 23515.246} C_VEL
LIN {X 0,Y 506.219,Z 1032.477,A -85,B 0,C 180,E1 23512.776,E2 23512.776} C_VEL
LIN {X 0,Y 502.759,Z 1046.042,A -85,B 0,C 180,E1 23510.732,E2 23510.732} C_VEL
LIN {X 0,Y 499.561,Z 1058.854,A -85,B 0,C 180,E1 23508.556,E2 23508.556} C_VEL
LIN {X 0,Y 496.079,Z 1073.557,A -85,B 0,C 180,E1 23505.669,E2 23505.669} C_VEL
LIN {X 0,Y 493.724,Z 1084.198,A -85,B 0,C 180,E1 23503.229,E2 23503.229} C_VEL
LIN {X 0,Y 491.882,Z 1093.51,A -85,B 0,C 180,E1 23500.778,E2 23500.778} C_VEL
LIN {X 0,Y 490.154,Z 1103.628,A -85,B 0,C 180,E1 23497.619,E2 23497.619} C_VEL
LIN {X 0,Y 489.22,Z 1110.407,A -85,B 0,C 180,E1 23495.042,E2 23495.042} C_VEL
LIN {X 0,Y 488.628,Z 1115.787,A -85,B 0,C 180,E1 23492.58,E2 23492.58} C_VEL
LIN {X 0,Y 488.233,Z 1120.894,A -85,B 0,C 180,E1 23489.648,E2 23489.648} C_VEL
LIN {X 0,Y 488.047,Z 1124.36,A -85,B 0,C 180,E1 23486.711,E2 23486.711} C_VEL
LIN {X 0,Y 487.996,Z 1126.22,A -85,B 0,C 180,E1 23484.238,E2 23484.238} C_VEL
LIN {X 0,Y 487.998,Z 1127.08,A -85,B 0,C 180,E1 23481.752,E2 23481.752} C_VEL
LIN {X 0,Y 487.994,Z 1126.844,A -85,B 0,C 180,E1 23478.776,E2 23478.776} C_VEL
LIN {X 0,Y 488.036,Z 1125.035,A -85,B 0,C 180,E1 23475.889,E2 23475.889} C_VEL
LIN {X 0,Y 488.146,Z 1122.499,A -85,B 0,C 180,E1 23473.458,E2 23473.458} C_VEL
LIN {X 0,Y 488.396,Z 1118.742,A -85,B 0,C 180,E1 23470.879,E2 23470.879} C_VEL
LIN {X 0,Y 488.988,Z 1112.74,A -85,B 0,C 180,E1 23467.773,E2 23467.773} C_VEL
LIN {X 0,Y 489.897,Z 1105.792,A -85,B 0,C 180,E1 23464.988,E2 23464.988} C_VEL
LIN {X 0,Y 491.121,Z 1098.335,A -85,B 0,C 180,E1 23462.475,E2 23462.475} C_VEL
